LIN {X 0,Y 580.292,Z 680.195,A -85,B 0,C 180,E1 -1968.827,E2 -1968.827} C_VEL
LIN {X 0,Y 580.317,Z 680.194,A -85,B 0,C 180,E1 -1971.644,E2 -1971.644} C_VEL
LIN {X 0,Y 580.327,Z 680.195,A -85,B 0,C 180,E1 -1974.44,E2 -1974.44} C_VEL
LIN {X 0,Y 580.324,Z 680.19,A -85,B 0,C 180,E1 -1977.223,E2 -1977.223} C_VEL
LIN {X 0,Y 580.334,Z 680.194,A -85,B 0,C 180,E1 -1980,E2 -1980} C_VEL
LIN {X 0,Y 580.338,Z 680.194,A -85,B 0,C 180,E1 -1982.777,E2 -1982.777} C_VEL
LIN {X 0,Y 580.312,Z 680.192,A -85,B 0,C 180,E1 -1985.56,E2 -1985.56} C_VEL
LIN {X 0,Y 580.321,Z 680.196,A -85,B 0,C 180,E1 -1988.356,E2 -1988.356} C_VEL
LIN {X 0,Y 580.322,Z 680.194,A -85,B 0,C 180,E1 -1991.209,E2 -1991.209} C_VEL
LIN {X 0,Y 580.297,Z 680.196,A -85,B 0,C 180,E1 -1994.337,E2 -1994.337} C_VEL
LIN {X 0,Y 580.3,Z 680.203,A -85,B 0,C 180,E1 -1996.914,E2 -1996.914} C_VEL
LIN {X 0,Y 580.291,Z 680.195,A -85,B 0,C 180,E1 -1999.823,E2 -1999.823} C_VEL
LIN {X 0,Y 580.269,Z 680.204,A -85,B 0,C 180,E1 -2001.343,E2 -2001.343} C_VEL
LIN {X 0,Y 579.573,Z 680.286,A -85,B 0,C 180,E1 -2001.923,E2 -2001.923} C_VEL
LIN {X 0,Y 576.697,Z 680.647,A -85,B 0,C 180,E1 -2002.862,E2 -2002.862} C_VEL
LIN {X 0,Y 574.296,Z 680.944,A -85,B 0,C 180,E1 -2003.619,E2 -2003.619} C_VEL
LIN {X 0,Y 573.284,Z 681.066,A -85,B 0,C 180,E1 -2004.203,E2 -2004.203} C_VEL
LIN {X 0,Y 573.211,Z 681.076,A -85,B 0,C 180,E1 -2004.4,E2 -2004.4} C_VEL
LIN {X 0,Y 573.238,Z 681.079,A -85,B 0,C 180,E1 -2006.977,E2 -2006.977} C_VEL
LIN {X 0,Y 573.235,Z 681.084,A -85,B 0,C 180,E1 -2009.489,E2 -2009.489} C_VEL
LIN {X 0,Y 573.244,Z 681.072,A -85,B 0,C 180,E1 -2012.646,E2 -2012.646} C_VEL
LIN {X 0,Y 573.243,Z 681.077,A -85,B 0,C 180,E1 -2015.186,E2 -2015.186} C_VEL
LIN {X 0,Y 573.228,Z 681.083,A -85,B 0,C 180,E1 -2017.809,E2 -2017.809} C_VEL
LIN {X 0,Y 573.237,Z 681.075,A -85,B 0,C 180,E1 -2020.526,E2 -2020.526} C_VEL
LIN {X 0,Y 573.231,Z 681.077,A -85,B 0,C 180,E1 -2023.36,E2 -2023.36} C_VEL
LIN {X 0,Y 573.229,Z 681.08,A -85,B 0,C 180,E1 -2026.333,E2 -2026.333} C_VEL
LIN {X 0,Y 573.22,Z 681.08,A -85,B 0,C 180,E1 -2028.544,E2 -2028.544} C_VEL
LIN {X 0,Y 573.301,Z 681.29,A -85,B 0,C 180,E1 -2031.465,E2 -2031.465} C_VEL
LIN {X 0,Y 573.493,Z 682.25,A -85,B 0,C 180,E1 -2031.564,E2 -2031.564} C_VEL
LIN {X 0,Y 574.016,Z 685.356,A -85,B 0,C 180,E1 -2031.626,E2 -2031.626} C_VEL
LIN {X 0,Y 573.888,Z 762.761,A -85,B 0,C 180,E1 -2032.619,E2 -2032.619} C_VEL
LIN {X 0,Y 573.797,Z 776.245,A -85,B 0,C 180,E1 -2032.945,E2 -2032.945} C_VEL
LIN {X 0,Y 573.673,Z 788.533,A -85,B 0,C 180,E1 -2033.385,E2 -2033.385} C_VEL
LIN {X 0,Y 573.574,Z 800.656,A -85,B 0,C 180,E1 -2033.976,E2 -2033.976} C_VEL
LIN {X 0,Y 573.428,Z 812.525,A -85,B 0,C 180,E1 -2034.722,E2 -2034.722} C_VEL
LIN {X 0,Y 573.348,Z 822.555,A -85,B 0,C 180,E1 -2035.512,E2 -2035.512} C_VEL
LIN {X 0,Y 573.187,Z 832.534,A -85,B 0,C 180,E1 -2036.488,E2 -2036.488} C_VEL
LIN {X 0,Y 573.17,Z 839.774,A -85,B 0,C 180,E1 -2037.351,E2 -2037.351} C_VEL
LIN {X 0,Y 573.102,Z 846.922,A -85,B 0,C 180,E1 -2038.384,E2 -2038.384} C_VEL
LIN {X 0,Y 573.027,Z 853.016,A -85,B 0,C 180,E1 -2039.48,E2 -2039.48} C_VEL
LIN {X 0,Y 573.024,Z 857.961,A -85,B 0,C 180,E1 -2040.622,E2 -2040.622} C_VEL
LIN {X 0,Y 572.974,Z 860.64,A -85,B 0,C 180,E1 -2041.423,E2 -2041.423} C_VEL
LIN {X 0,Y 572.963,Z 862.779,A -85,B 0,C 180,E1 -2042.219,E2 -2042.219} C_VEL
LIN {X 0,Y 572.961,Z 865.101,A -85,B 0,C 180,E1 -2043.564,E2 -2043.564} C_VEL
LIN {X 0,Y 572.939,Z 865.901,A -85,B 0,C 180,E1 -2044.576,E2 -2044.576} C_VEL
LIN {X 0,Y 572.951,Z 865.938,A -85,B 0,C 180,E1 -2045.353,E2 -2045.353} C_VEL
LIN {X 0,Y 572.926,Z 865.53,A -85,B 0,C 180,E1 -2046.122,E2 -2046.122} C_VEL
LIN {X 0,Y 572.952,Z 864.563,A -85,B 0,C 180,E1 -2046.923,E2 -2046.923} C_VEL
LIN {X 0,Y 572.945,Z 863.24,A -85,B 0,C 180,E1 -2047.652,E2 -2047.652} C_VEL
LIN {X 0,Y 572.989,Z 860.305,A -85,B 0,C 180,E1 -2048.778,E2 -2048.778} C_VEL
LIN {X 0,Y 573.03,Z 856.166,A -85,B 0,C 180,E1 -2049.917,E2 -2049.917} C_VEL
LIN {X 0,Y 573.072,Z 850.484,A -85,B 0,C 180,E1 -2051.099,E2 -2051.099} C_VEL
LIN {X 0,Y 573.119,Z 844.051,A -85,B 0,C 180,E1 -2052.149,E2 -2052.149} C_VEL
LIN {X 0,Y 573.174,Z 836.754,A -85,B 0,C 180,E1 -2053.118,E2 -2053.118} C_VEL
LIN {X 0,Y 573.266,Z 826.991,A -85,B 0,C 180,E1 -2054.172,E2 -2054.172} C_VEL
LIN {X 0,Y 573.368,Z 817.537,A -85,B 0,C 180,E1 -2054.994,E2 -2054.994} C_VEL
LIN {X 0,Y 573.504,Z 807.239,A -85,B 0,C 180,E1 -2055.723,E2 -2055.723} C_VEL
LIN {X 0,Y 573.606,Z 796.002,A -85,B 0,C 180,E1 -2056.359,E2 -2056.359} C_VEL
LIN {X 0,Y 573.724,Z 783.527,A -85,B 0,C 180,E1 -2056.903,E2 -2056.903} C_VEL
LIN {X 0,Y 573.833,Z 770.218,A -85,B 0,C 180,E1 -2057.31,E2 -2057.31} C_VEL
LIN {X 0,Y 573.914,Z 757.259,A -85,B 0,C 180,E1 -2057.559,E2 -2057.559} C_VEL
LIN {X 0,Y 573.909,Z 683.635,A -85,B 0,C 180,E1 -2058.488,E2 -2058.488} C_VEL
LIN {X 0,Y 573.375,Z 681.682,A -85,B 0,C 180,E1 -2058.567,E2 -2058.567} C_VEL
LIN {X 0,Y 573.274,Z 681.113,A -85,B 0,C 180,E1 -2058.689,E2 -2058.689} C_VEL
LIN {X 0,Y 573.245,Z 681.078,A -85,B 0,C 180,E1 -2061.541,E2 -2061.541} C_VEL
LIN {X 0,Y 573.267,Z 681.076,A -85,B 0,C 180,E1 -2064.373,E2 -2064.373} C_VEL
LIN {X 0,Y 573.309,Z 681.071,A -85,B 0,C 180,E1 -2067.893,E2 -2067.893} C_VEL
LIN {X 0,Y 573.319,Z 681.071,A -85,B 0,C 180,E1 -2070.001,E2 -2070.001} C_VEL
LIN {X 0,Y 573.279,Z 681.072,A -85,B 0,C 180,E1 -2072.812,E2 -2072.812} C_VEL
LIN {X 0,Y 573.257,Z 681.072,A -85,B 0,C 180,E1 -2075.63,E2 -2075.63} C_VEL
LIN {X 0,Y 573.237,Z 681.084,A -85,B 0,C 180,E1 -2078.461,E2 -2078.461} C_VEL
LIN {X 0,Y 573.239,Z 681.074,A -85,B 0,C 180,E1 -2081.314,E2 -2081.314} C_VEL
LIN {X 0,Y 573.264,Z 681.076,A -85,B 0,C 180,E1 -2084.415,E2 -2084.415} C_VEL
LIN {X 0,Y 573.223,Z 681.08,A -85,B 0,C 180,E1 -2087.114,E2 -2087.114} C_VEL
LIN {X 0,Y 573.205,Z 681.076,A -85,B 0,C 180,E1 -2090.079,E2 -2090.079} C_VEL
LIN {X 0,Y 573.218,Z 681.078,A -85,B 0,C 180,E1 -2092.34,E2 -2092.34} C_VEL
LIN {X 0,Y 573.196,Z 681.081,A -85,B 0,C 180,E1 -2095.414,E2 -2095.414} C_VEL
LIN {X 0,Y 573.2,Z 681.077,A -85,B 0,C 180,E1 -2098.018,E2 -2098.018} C_VEL
LIN {X 0,Y 573.201,Z 681.083,A -85,B 0,C 180,E1 -2100.877,E2 -2100.877} C_VEL
LIN {X 0,Y 573.195,Z 681.082,A -85,B 0,C 180,E1 -2103.513,E2 -2103.513} C_VEL
LIN {X 0,Y 573.181,Z 681.079,A -85,B 0,C 180,E1 -2106.055,E2 -2106.055} C_VEL
LIN {X 0,Y 573.177,Z 681.081,A -85,B 0,C 180,E1 -2108.708,E2 -2108.708} C_VEL
LIN {X 0,Y 573.194,Z 681.089,A -85,B 0,C 180,E1 -2111.588,E2 -2111.588} C_VEL
LIN {X 0,Y 573.207,Z 681.078,A -85,B 0,C 180,E1 -2114.337,E2 -2114.337} C_VEL
LIN {X 0,Y 573.213,Z 681.081,A -85,B 0,C 180,E1 -2117.363,E2 -2117.363} C_VEL
LIN {X 0,Y 573.224,Z 681.076,A -85,B 0,C 180,E1 -2120.572,E2 -2120.572} C_VEL
LIN {X 0,Y 573.183,Z 681.081,A -85,B 0,C 180,E1 -2123.072,E2 -2123.072} C_VEL
LIN {X 0,Y 573.242,Z 681.079,A -85,B 0,C 180,E1 -2125.669,E2 -2125.669} C_VEL
LIN {X 0,Y 573.21,Z 681.087,A -85,B 0,C 180,E1 -2128.182,E2 -2128.182} C_VEL
LIN {X 0,Y 573.221,Z 681.08,A -85,B 0,C 180,E1 -2130.631,E2 -2130.631} C_VEL
LIN {X 0,Y 573.257,Z 681.217,A -85,B 0,C 180,E1 -2133.443,E2 -2133.443} C_VEL
LIN {X 0,Y 573.405,Z 682.037,A -85,B 0,C 180,E1 -2133.552,E2 -2133.552} C_VEL
LIN {X 0,Y 574.019,Z 683.936,A -85,B 0,C 180,E1 -2133.608,E2 -2133.608} C_VEL
LIN {X 0,Y 573.874,Z 761.452,A -85,B 0,C 180,E1 -2134.595,E2 -2134.595} C_VEL
LIN {X 0,Y 573.817,Z 774.103,A -85,B 0,C 180,E1 -2134.885,E2 -2134.885} C_VEL
LIN {X 0,Y 573.684,Z 785.769,A -85,B 0,C 180,E1 -2135.278,E2 -2135.278} C_VEL
LIN {X 0,Y 573.596,Z 796.622,A -85,B 0,C 180,E1 -2135.766,E2 -2135.766} C_VEL
LIN {X 0,Y 573.486,Z 806.696,A -85,B 0,C 180,E1 -2136.337,E2 -2136.337} C_VEL
LIN {X 0,Y 573.375,Z 816.262,A -85,B 0,C 180,E1 -2137.002,E2 -2137.002} C_VEL
LIN {X 0,Y 573.273,Z 826.276,A -85,B 0,C 180,E1 -2137.853,E2 -2137.853} C_VEL
LIN {X 0,Y 573.166,Z 836.526,A -85,B 0,C 180,E1 -2138.943,E2 -2138.943} C_VEL
LIN {X 0,Y 573.09,Z 843.894,A -85,B 0,C 180,E1 -2139.917,E2 -2139.917} C_VEL
LIN {X 0,Y 573.05,Z 851.003,A -85,B 0,C 180,E1 -2141.096,E2 -2141.096} C_VEL
LIN {X 0,Y 572.995,Z 856.009,A -85,B 0,C 180,E1 -2142.143,E2 -2142.143} C_VEL
LIN {X 0,Y 572.999,Z 859.538,A -85,B 0,C 180,E1 -2143.078,E2 -2143.078} C_VEL
LIN {X 0,Y 572.934,Z 863.018,A -85,B 0,C 180,E1 -2144.343,E2 -2144.343} C_VEL
LIN {X 0,Y 572.948,Z 865.26,A -85,B 0,C 180,E1 -2145.709,E2 -2145.709} C_VEL
LIN {X 0,Y 572.971,Z 865.85,A -85,B 0,C 180,E1 -2146.523,E2 -2146.523} C_VEL
LIN {X 0,Y 572.946,Z 865.962,A -85,B 0,C 180,E1 -2147.244,E2 -2147.244} C_VEL
LIN {X 0,Y 572.948,Z 865.641,A -85,B 0,C 180,E1 -2147.964,E2 -2147.964} C_VEL
LIN {X 0,Y 572.986,Z 863.757,A -85,B 0,C 180,E1 -2149.398,E2 -2149.398} C_VEL
LIN {X 0,Y 572.985,Z 861.23,A -85,B 0,C 180,E1 -2150.469,E2 -2150.469} C_VEL
LIN {X 0,Y 573.022,Z 857.69,A -85,B 0,C 180,E1 -2151.536,E2 -2151.536} C_VEL
LIN {X 0,Y 573.028,Z 853.051,A -85,B 0,C 180,E1 -2152.601,E2 -2152.601} C_VEL
LIN {X 0,Y 573.057,Z 847.179,A -85,B 0,C 180,E1 -2153.663,E2 -2153.663} C_VEL
LIN {X 0,Y 573.1,Z 839.878,A -85,B 0,C 180,E1 -2154.723,E2 -2154.723} C_VEL
LIN {X 0,Y 573.22,Z 832.446,A -85,B 0,C 180,E1 -2155.605,E2 -2155.605} C_VEL
LIN {X 0,Y 573.281,Z 825.479,A -85,B 0,C 180,E1 -2156.31,E2 -2156.31} C_VEL
LIN {X 0,Y 573.401,Z 816.075,A -85,B 0,C 180,E1 -2157.102,E2 -2157.102} C_VEL
LIN {X 0,Y 573.518,Z 805.856,A -85,B 0,C 180,E1 -2157.805,E2 -2157.805} C_VEL
LIN {X 0,Y 573.578,Z 794.739,A -85,B 0,C 180,E1 -2158.42,E2 -2158.42} C_VEL
LIN {X 0,Y 573.758,Z 783.44,A -85,B 0,C 180,E1 -2158.903,E2 -2158.903} C_VEL
LIN {X 0,Y 573.836,Z 768.97,A -85,B 0,C 180,E1 -2159.342,E2 -2159.342} C_VEL
LIN {X 0,Y 573.918,Z 755.563,A -85,B 0,C 180,E1 -2159.583,E2 -2159.583} C_VEL
LIN {X 0,Y 574.036,Z 683.885,A -85,B 0,C 180,E1 -2160.482,E2 -2160.482} C_VEL
LIN {X 0,Y 573.443,Z 681.868,A -85,B 0,C 180,E1 -2160.548,E2 -2160.548} C_VEL
LIN {X 0,Y 573.329,Z 681.115,A -85,B 0,C 180,E1 -2160.702,E2 -2160.702} C_VEL
LIN {X 0,Y 573.303,Z 681.068,A -85,B 0,C 180,E1 -2162.811,E2 -2162.811} C_VEL
LIN {X 0,Y 573.291,Z 681.072,A -85,B 0,C 180,E1 -2165.628,E2 -2165.628} C_VEL
LIN {X 0,Y 573.259,Z 681.077,A -85,B 0,C 180,E1 -2168.46,E2 -2168.46} C_VEL
LIN {X 0,Y 573.279,Z 681.069,A -85,B 0,C 180,E1 -2171.312,E2 -2171.312} C_VEL
LIN {X 0,Y 573.288,Z 681.077,A -85,B 0,C 180,E1 -2174.424,E2 -2174.424} C_VEL
LIN {X 0,Y 573.262,Z 681.072,A -85,B 0,C 180,E1 -2177.111,E2 -2177.111} C_VEL
LIN {X 0,Y 573.247,Z 681.076,A -85,B 0,C 180,E1 -2180.077,E2 -2180.077} C_VEL
LIN {X 0,Y 573.237,Z 681.08,A -85,B 0,C 180,E1 -2182.338,E2 -2182.338} C_VEL
LIN {X 0,Y 573.252,Z 681.073,A -85,B 0,C 180,E1 -2185.41,E2 -2185.41} C_VEL
LIN {X 0,Y 573.234,Z 681.081,A -85,B 0,C 180,E1 -2188.565,E2 -2188.565} C_VEL
LIN {X 0,Y 573.23,Z 681.083,A -85,B 0,C 180,E1 -2190.993,E2 -2190.993} C_VEL
LIN {X 0,Y 573.247,Z 681.075,A -85,B 0,C 180,E1 -2193.52,E2 -2193.52} C_VEL
LIN {X 0,Y 573.22,Z 681.076,A -85,B 0,C 180,E1 -2196.051,E2 -2196.051} C_VEL
LIN {X 0,Y 573.244,Z 681.077,A -85,B 0,C 180,E1 -2198.702,E2 -2198.702} C_VEL
LIN {X 0,Y 573.233,Z 681.079,A -85,B 0,C 180,E1 -2201.592,E2 -2201.592} C_VEL
LIN {X 0,Y 573.228,Z 681.075,A -85,B 0,C 180,E1 -2204.334,E2 -2204.334} C_VEL
LIN {X 0,Y 573.245,Z 681.083,A -85,B 0,C 180,E1 -2207.358,E2 -2207.358} C_VEL
LIN {X 0,Y 573.241,Z 681.073,A -85,B 0,C 180,E1 -2210.391,E2 -2210.391} C_VEL
LIN {X 0,Y 573.238,Z 681.076,A -85,B 0,C 180,E1 -2213.075,E2 -2213.075} C_VEL
LIN {X 0,Y 573.26,Z 681.081,A -85,B 0,C 180,E1 -2215.67,E2 -2215.67} C_VEL
LIN {X 0,Y 573.245,Z 681.078,A -85,B 0,C 180,E1 -2218.184,E2 -2218.184} C_VEL
LIN {X 0,Y 573.265,Z 681.074,A -85,B 0,C 180,E1 -2220.633,E2 -2220.633} C_VEL
LIN {X 0,Y 573.257,Z 681.272,A -85,B 0,C 180,E1 -2222.629,E2 -2222.629} C_VEL
LIN {X 0,Y 574.935,Z 688.635,A -85,B 0,C 180,E1 -2223.592,E2 -2223.592} C_VEL
LIN {X 0,Y 574.576,Z 711.379,A -85,B 0,C 180,E1 -2226.193,E2 -2226.193} C_VEL
LIN {X 0,Y 574.209,Z 738.275,A -85,B 0,C 180,E1 -2229.209,E2 -2229.209} C_VEL
LIN {X 0,Y 573.871,Z 765.171,A -85,B 0,C 180,E1 -2232.171,E2 -2232.171} C_VEL
LIN {X 0,Y 573.599,Z 792.067,A -85,B 0,C 180,E1 -2235.089,E2 -2235.089} C_VEL
LIN {X 0,Y 573.536,Z 801.874,A -85,B 0,C 180,E1 -2236.129,E2 -2236.129} C_VEL
LIN {X 0,Y 574.037,Z 807.642,A -85,B 0,C 180,E1 -2236.232,E2 -2236.232} C_VEL
LIN {X 0,Y 573.876,Z 911.896,A -85,B 0,C 180,E1 -2237.556,E2 -2237.556} C_VEL
LIN {X 0,Y 573.832,Z 924.424,A -85,B 0,C 180,E1 -2237.847,E2 -2237.847} C_VEL
LIN {X 0,Y 573.708,Z 936.891,A -85,B 0,C 180,E1 -2238.275,E2 -2238.275} C_VEL
LIN {X 0,Y 573.612,Z 948.42,A -85,B 0,C 180,E1 -2238.809,E2 -2238.809} C_VEL
LIN {X 0,Y 573.475,Z 959.899,A -85,B 0,C 180,E1 -2239.496,E2 -2239.496} C_VEL
LIN {X 0,Y 573.345,Z 970.527,A -85,B 0,C 180,E1 -2240.296,E2 -2240.296} C_VEL
LIN {X 0,Y 573.238,Z 980.036,A -85,B 0,C 180,E1 -2241.184,E2 -2241.184} C_VEL
LIN {X 0,Y 573.161,Z 987.952,A -85,B 0,C 180,E1 -2242.07,E2 -2242.07} C_VEL
LIN {X 0,Y 573.076,Z 995.935,A -85,B 0,C 180,E1 -2243.183,E2 -2243.183} C_VEL
LIN {X 0,Y 573.07,Z 1002.675,A -85,B 0,C 180,E1 -2244.369,E2 -2244.369} C_VEL
LIN {X 0,Y 573.028,Z 1007.368,A -85,B 0,C 180,E1 -2245.426,E2 -2245.426} C_VEL
LIN {X 0,Y 573.022,Z 1010.954,A -85,B 0,C 180,E1 -2246.483,E2 -2246.483} C_VEL
LIN {X 0,Y 572.959,Z 1012.806,A -85,B 0,C 180,E1 -2247.187,E2 -2247.187} C_VEL
LIN {X 0,Y 572.938,Z 1014.198,A -85,B 0,C 180,E1 -2247.89,E2 -2247.89} C_VEL
LIN {X 0,Y 572.94,Z 1015.784,A -85,B 0,C 180,E1 -2249.296,E2 -2249.296} C_VEL
LIN {X 0,Y 572.938,Z 1016,A -85,B 0,C 180,E1 -2249.999,E2 -2249.999} C_VEL
LIN {X 0,Y 572.946,Z 1015.187,A -85,B 0,C 180,E1 -2251.405,E2 -2251.405} C_VEL
LIN {X 0,Y 572.938,Z 1014.202,A -85,B 0,C 180,E1 -2252.108,E2 -2252.108} C_VEL
LIN {X 0,Y 572.959,Z 1012.812,A -85,B 0,C 180,E1 -2252.811,E2 -2252.811} C_VEL
LIN {X 0,Y 573.014,Z 1009.899,A -85,B 0,C 180,E1 -2253.867,E2 -2253.867} C_VEL
LIN {X 0,Y 572.962,Z 1005.954,A -85,B 0,C 180,E1 -2254.925,E2 -2254.925} C_VEL
LIN {X 0,Y 573.067,Z 999.883,A -85,B 0,C 180,E1 -2256.159,E2 -2256.159} C_VEL
LIN {X 0,Y 573.118,Z 993.245,A -85,B 0,C 180,E1 -2257.22,E2 -2257.22} C_VEL
LIN {X 0,Y 573.191,Z 985,A -85,B 0,C 180,E1 -2258.282,E2 -2258.282} C_VEL
LIN {X 0,Y 573.319,Z 974.613,A -85,B 0,C 180,E1 -2259.347,E2 -2259.347} C_VEL
LIN {X 0,Y 573.43,Z 964.943,A -85,B 0,C 180,E1 -2260.146,E2 -2260.146} C_VEL
LIN {X 0,Y 573.552,Z 954.369,A -85,B 0,C 180,E1 -2260.857,E2 -2260.857} C_VEL
LIN {X 0,Y 573.685,Z 942.023,A -85,B 0,C 180,E1 -2261.504,E2 -2261.504} C_VEL
LIN {X 0,Y 573.737,Z 930.208,A -85,B 0,C 180,E1 -2261.973,E2 -2261.973} C_VEL
LIN {X 0,Y 573.842,Z 917.568,A -85,B 0,C 180,E1 -2262.33,E2 -2262.33} C_VEL
LIN {X 0,Y 573.946,Z 904.402,A -85,B 0,C 180,E1 -2262.552,E2 -2262.552} C_VEL
LIN {X 0,Y 573.986,Z 805.242,A -85,B 0,C 180,E1 -2263.8,E2 -2263.8} C_VEL
LIN {X 0,Y 573.534,Z 801.904,A -85,B 0,C 180,E1 -2263.869,E2 -2263.869} C_VEL
LIN {X 0,Y 573.769,Z 775.277,A -85,B 0,C 180,E1 -2266.728,E2 -2266.728} C_VEL
LIN {X 0,Y 574.121,Z 746.574,A -85,B 0,C 180,E1 -2269.871,E2 -2269.871} C_VEL
LIN {X 0,Y 574.399,Z 721.485,A -85,B 0,C 180,E1 -2272.668,E2 -2272.668} C_VEL
LIN {X 0,Y 574.808,Z 699.068,A -85,B 0,C 180,E1 -2275.207,E2 -2275.207} C_VEL
LIN {X 0,Y 574.941,Z 688.649,A -85,B 0,C 180,E1 -2276.406,E2 -2276.406} C_VEL
LIN {X 0,Y 573.258,Z 681.194,A -85,B 0,C 180,E1 -2277.394,E2 -2277.394} C_VEL
LIN {X 0,Y 573.243,Z 681.082,A -85,B 0,C 180,E1 -2280.175,E2 -2280.175} C_VEL
LIN {X 0,Y 573.249,Z 681.078,A -85,B 0,C 180,E1 -2282.644,E2 -2282.644} C_VEL
LIN {X 0,Y 573.201,Z 681.079,A -85,B 0,C 180,E1 -2285.187,E2 -2285.187} C_VEL
LIN {X 0,Y 573.228,Z 681.076,A -85,B 0,C 180,E1 -2287.806,E2 -2287.806} C_VEL
LIN {X 0,Y 573.237,Z 681.083,A -85,B 0,C 180,E1 -2290.524,E2 -2290.524} C_VEL
LIN {X 0,Y 573.232,Z 681.075,A -85,B 0,C 180,E1 -2293.358,E2 -2293.358} C_VEL
LIN {X 0,Y 573.248,Z 681.075,A -85,B 0,C 180,E1 -2296.329,E2 -2296.329} C_VEL
LIN {X 0,Y 573.266,Z 681.071,A -85,B 0,C 180,E1 -2299.477,E2 -2299.477} C_VEL
LIN {X 0,Y 573.228,Z 681.075,A -85,B 0,C 180,E1 -2302.192,E2 -2302.192} C_VEL
LIN {X 0,Y 573.259,Z 681.075,A -85,B 0,C 180,E1 -2304.816,E2 -2304.816} C_VEL
LIN {X 0,Y 573.244,Z 681.081,A -85,B 0,C 180,E1 -2307.354,E2 -2307.354} C_VEL
LIN {X 0,Y 573.243,Z 681.073,A -85,B 0,C 180,E1 -2310.51,E2 -2310.51} C_VEL
LIN {X 0,Y 573.253,Z 681.076,A -85,B 0,C 180,E1 -2313.024,E2 -2313.024} C_VEL
LIN {X 0,Y 573.264,Z 681.079,A -85,B 0,C 180,E1 -2315.366,E2 -2315.366} C_VEL
LIN {X 0,Y 573.218,Z 681.075,A -85,B 0,C 180,E1 -2318.419,E2 -2318.419} C_VEL
LIN {X 0,Y 573.266,Z 681.07,A -85,B 0,C 180,E1 -2320.728,E2 -2320.728} C_VEL
LIN {X 0,Y 573.235,Z 681.081,A -85,B 0,C 180,E1 -2323.621,E2 -2323.621} C_VEL
LIN {X 0,Y 573.262,Z 681.081,A -85,B 0,C 180,E1 -2325.807,E2 -2325.807} C_VEL
LIN {X 0,Y 573.25,Z 681.072,A -85,B 0,C 180,E1 -2328.745,E2 -2328.745} C_VEL
LIN {X 0,Y 573.273,Z 681.07,A -85,B 0,C 180,E1 -2331.54,E2 -2331.54} C_VEL
LIN {X 0,Y 573.293,Z 681.073,A -85,B 0,C 180,E1 -2334.372,E2 -2334.372} C_VEL
LIN {X 0,Y 573.292,Z 681.066,A -85,B 0,C 180,E1 -2337.189,E2 -2337.189} C_VEL
LIN {X 0,Y 573.304,Z 681.069,A -85,B 0,C 180,E1 -2340,E2 -2340} C_VEL
LIN {X 0,Y 573.303,Z 681.07,A -85,B 0,C 180,E1 -2342.811,E2 -2342.811} C_VEL
LIN {X 0,Y 573.278,Z 681.068,A -85,B 0,C 180,E1 -2345.628,E2 -2345.628} C_VEL
LIN {X 0,Y 573.278,Z 681.076,A -85,B 0,C 180,E1 -2348.46,E2 -2348.46} C_VEL
LIN {X 0,Y 573.288,Z 681.069,A -85,B 0,C 180,E1 -2351.312,E2 -2351.312} C_VEL
LIN {X 0,Y 573.264,Z 681.074,A -85,B 0,C 180,E1 -2354.423,E2 -2354.423} C_VEL
LIN {X 0,Y 573.246,Z 681.081,A -85,B 0,C 180,E1 -2357.112,E2 -2357.112} C_VEL
LIN {X 0,Y 573.238,Z 681.073,A -85,B 0,C 180,E1 -2360.077,E2 -2360.077} C_VEL
LIN {X 0,Y 573.224,Z 681.084,A -85,B 0,C 180,E1 -2363.1,E2 -2363.1} C_VEL
LIN {X 0,Y 573.211,Z 681.076,A -85,B 0,C 180,E1 -2364.4,E2 -2364.4} C_VEL
LIN {X 0,Y 572.573,Z 681.162,A -85,B 0,C 180,E1 -2364.987,E2 -2364.987} C_VEL
LIN {X 0,Y 569.74,Z 681.521,A -85,B 0,C 180,E1 -2365.938,E2 -2365.938} C_VEL
LIN {X 0,Y 567.325,Z 681.825,A -85,B 0,C 180,E1 -2366.704,E2 -2366.704} C_VEL
LIN {X 0,Y 566.279,Z 681.951,A -85,B 0,C 180,E1 -2367.296,E2 -2367.296} C_VEL
LIN {X 0,Y 566.191,Z 681.958,A -85,B 0,C 180,E1 -2367.496,E2 -2367.496} C_VEL
LIN {X 0,Y 566.19,Z 681.957,A -85,B 0,C 180,E1 -2369.77,E2 -2369.77} C_VEL
LIN {X 0,Y 566.194,Z 681.95,A -85,B 0,C 180,E1 -2372.431,E2 -2372.431} C_VEL
LIN {X 0,Y 566.191,Z 681.953,A -85,B 0,C 180,E1 -2374.993,E2 -2374.993} C_VEL
LIN {X 0,Y 566.188,Z 681.959,A -85,B 0,C 180,E1 -2377.462,E2 -2377.462} C_VEL
LIN {X 0,Y 566.199,Z 681.955,A -85,B 0,C 180,E1 -2380.2,E2 -2380.2} C_VEL
LIN {X 0,Y 566.194,Z 681.951,A -85,B 0,C 180,E1 -2383.055,E2 -2383.055} C_VEL
LIN {X 0,Y 566.187,Z 681.96,A -85,B 0,C 180,E1 -2386.051,E2 -2386.051} C_VEL
LIN {X 0,Y 566.198,Z 681.953,A -85,B 0,C 180,E1 -2389.216,E2 -2389.216} C_VEL
LIN {X 0,Y 566.254,Z 682.179,A -85,B 0,C 180,E1 -2391.306,E2 -2391.306} C_VEL
LIN {X 0,Y 566.569,Z 683.524,A -85,B 0,C 180,E1 -2391.42,E2 -2391.42} C_VEL
LIN {X 0,Y 567.115,Z 685.653,A -85,B 0,C 180,E1 -2391.463,E2 -2391.463} C_VEL
LIN {X 0,Y 566.971,Z 762.537,A -85,B 0,C 180,E1 -2392.46,E2 -2392.46} C_VEL
LIN {X 0,Y 566.859,Z 776.007,A -85,B 0,C 180,E1 -2392.787,E2 -2392.787} C_VEL
LIN {X 0,Y 566.736,Z 787.432,A -85,B 0,C 180,E1 -2393.195,E2 -2393.195} C_VEL
LIN {X 0,Y 566.625,Z 798.688,A -85,B 0,C 180,E1 -2393.728,E2 -2393.728} C_VEL
LIN {X 0,Y 566.498,Z 810.11,A -85,B 0,C 180,E1 -2394.425,E2 -2394.425} C_VEL
LIN {X 0,Y 566.311,Z 820.193,A -85,B 0,C 180,E1 -2395.191,E2 -2395.191} C_VEL
LIN {X 0,Y 566.213,Z 829.39,A -85,B 0,C 180,E1 -2396.046,E2 -2396.046} C_VEL
LIN {X 0,Y 566.05,Z 838.458,A -85,B 0,C 180,E1 -2397.08,E2 -2397.08} C_VEL
LIN {X 0,Y 566.041,Z 845.999,A -85,B 0,C 180,E1 -2398.152,E2 -2398.152} C_VEL
LIN {X 0,Y 565.956,Z 852.941,A -85,B 0,C 180,E1 -2399.395,E2 -2399.395} C_VEL
LIN {X 0,Y 565.93,Z 858.454,A -85,B 0,C 180,E1 -2400.708,E2 -2400.708} C_VEL
LIN {X 0,Y 565.868,Z 861.979,A -85,B 0,C 180,E1 -2401.862,E2 -2401.862} C_VEL
LIN {X 0,Y 565.844,Z 863.724,A -85,B 0,C 180,E1 -2402.643,E2 -2402.643} C_VEL
LIN {X 0,Y 565.856,Z 864.984,A -85,B 0,C 180,E1 -2403.442,E2 -2403.442} C_VEL
LIN {X 0,Y 565.829,Z 865.72,A -85,B 0,C 180,E1 -2404.234,E2 -2404.234} C_VEL
LIN {X 0,Y 565.838,Z 866,A -85,B 0,C 180,E1 -2405.054,E2 -2405.054} C_VEL
LIN {X 0,Y 565.825,Z 865.754,A -85,B 0,C 180,E1 -2405.804,E2 -2405.804} C_VEL
LIN {X 0,Y 565.833,Z 864.79,A -85,B 0,C 180,E1 -2406.8,E2 -2406.8} C_VEL
LIN {X 0,Y 565.854,Z 862.235,A -85,B 0,C 180,E1 -2408.125,E2 -2408.125} C_VEL
LIN {X 0,Y 565.898,Z 858.838,A -85,B 0,C 180,E1 -2409.272,E2 -2409.272} C_VEL
LIN {X 0,Y 565.973,Z 854.261,A -85,B 0,C 180,E1 -2410.412,E2 -2410.412} C_VEL
LIN {X 0,Y 565.988,Z 848.418,A -85,B 0,C 180,E1 -2411.541,E2 -2411.541} C_VEL
LIN {X 0,Y 566.061,Z 841.064,A -85,B 0,C 180,E1 -2412.665,E2 -2412.665} C_VEL
LIN {X 0,Y 566.194,Z 831.852,A -85,B 0,C 180,E1 -2413.784,E2 -2413.784} C_VEL
LIN {X 0,Y 566.267,Z 822.433,A -85,B 0,C 180,E1 -2414.709,E2 -2414.709} C_VEL
LIN {X 0,Y 566.408,Z 811.869,A -85,B 0,C 180,E1 -2415.544,E2 -2415.544} C_VEL
LIN {X 0,Y 566.593,Z 800.19,A -85,B 0,C 180,E1 -2416.278,E2 -2416.278} C_VEL
LIN {X 0,Y 566.733,Z 787.92,A -85,B 0,C 180,E1 -2416.875,E2 -2416.875} C_VEL
LIN {X 0,Y 566.879,Z 774.93,A -85,B 0,C 180,E1 -2417.334,E2 -2417.334} C_VEL
LIN {X 0,Y 566.952,Z 762.486,A -85,B 0,C 180,E1 -2417.631,E2 -2417.631} C_VEL
LIN {X 0,Y 567.037,Z 685.043,A -85,B 0,C 180,E1 -2418.636,E2 -2418.636} C_VEL
LIN {X 0,Y 566.368,Z 682.687,A -85,B 0,C 180,E1 -2418.714,E2 -2418.714} C_VEL
LIN {X 0,Y 566.215,Z 682.009,A -85,B 0,C 180,E1 -2418.84,E2 -2418.84} C_VEL
LIN {X 0,Y 566.196,Z 681.956,A -85,B 0,C 180,E1 -2421.435,E2 -2421.435} C_VEL
LIN {X 0,Y 566.238,Z 681.953,A -85,B 0,C 180,E1 -2424.303,E2 -2424.303} C_VEL
LIN {X 0,Y 566.279,Z 681.947,A -85,B 0,C 180,E1 -2427.867,E2 -2427.867} C_VEL
LIN {X 0,Y 566.288,Z 681.947,A -85,B 0,C 180,E1 -2430.001,E2 -2430.001} C_VEL
LIN {X 0,Y 566.245,Z 681.948,A -85,B 0,C 180,E1 -2432.847,E2 -2432.847} C_VEL
LIN {X 0,Y 566.228,Z 681.948,A -85,B 0,C 180,E1 -2435.7,E2 -2435.7} C_VEL
LIN {X 0,Y 566.19,Z 681.962,A -85,B 0,C 180,E1 -2438.567,E2 -2438.567} C_VEL
LIN {X 0,Y 566.195,Z 681.951,A -85,B 0,C 180,E1 -2441.456,E2 -2441.456} C_VEL
LIN {X 0,Y 566.219,Z 681.955,A -85,B 0,C 180,E1 -2444.498,E2 -2444.498} C_VEL
LIN {X 0,Y 566.176,Z 681.955,A -85,B 0,C 180,E1 -2447.333,E2 -2447.333} C_VEL
LIN {X 0,Y 566.178,Z 681.951,A -85,B 0,C 180,E1 -2449.583,E2 -2449.583} C_VEL
LIN {X 0,Y 566.187,Z 681.952,A -85,B 0,C 180,E1 -2451.864,E2 -2451.864} C_VEL
LIN {X 0,Y 566.152,Z 681.956,A -85,B 0,C 180,E1 -2454.184,E2 -2454.184} C_VEL
LIN {X 0,Y 566.165,Z 681.956,A -85,B 0,C 180,E1 -2456.649,E2 -2456.649} C_VEL
LIN {X 0,Y 566.141,Z 681.96,A -85,B 0,C 180,E1 -2459.66,E2 -2459.66} C_VEL
LIN {X 0,Y 566.176,Z 681.953,A -85,B 0,C 180,E1 -2462.425,E2 -2462.425} C_VEL
LIN {X 0,Y 566.152,Z 681.957,A -85,B 0,C 180,E1 -2464.985,E2 -2464.985} C_VEL
LIN {X 0,Y 566.182,Z 681.962,A -85,B 0,C 180,E1 -2467.463,E2 -2467.463} C_VEL
LIN {X 0,Y 566.161,Z 681.956,A -85,B 0,C 180,E1 -2470.204,E2 -2470.204} C_VEL
LIN {X 0,Y 566.137,Z 681.961,A -85,B 0,C 180,E1 -2473.061,E2 -2473.061} C_VEL
LIN {X 0,Y 566.14,Z 681.962,A -85,B 0,C 180,E1 -2476.056,E2 -2476.056} C_VEL
LIN {X 0,Y 566.134,Z 681.959,A -85,B 0,C 180,E1 -2478.856,E2 -2478.856} C_VEL
LIN {X 0,Y 566.158,Z 681.96,A -85,B 0,C 180,E1 -2481.45,E2 -2481.45} C_VEL
LIN {X 0,Y 566.135,Z 681.963,A -85,B 0,C 180,E1 -2484.306,E2 -2484.306} C_VEL
LIN {X 0,Y 566.165,Z 681.956,A -85,B 0,C 180,E1 -2486.894,E2 -2486.894} C_VEL
LIN {X 0,Y 566.161,Z 681.958,A -85,B 0,C 180,E1 -2489.406,E2 -2489.406} C_VEL
LIN {X 0,Y 566.133,Z 681.966,A -85,B 0,C 180,E1 -2491.853,E2 -2491.853} C_VEL
LIN {X 0,Y 566.195,Z 682.159,A -85,B 0,C 180,E1 -2493.297,E2 -2493.297} C_VEL
LIN {X 0,Y 566.489,Z 683.306,A -85,B 0,C 180,E1 -2493.414,E2 -2493.414} C_VEL
LIN {X 0,Y 567.125,Z 685.465,A -85,B 0,C 180,E1 -2493.461,E2 -2493.461} C_VEL
LIN {X 0,Y 566.962,Z 761.993,A -85,B 0,C 180,E1 -2494.452,E2 -2494.452} C_VEL
LIN {X 0,Y 566.853,Z 773.749,A -85,B 0,C 180,E1 -2494.723,E2 -2494.723} C_VEL
LIN {X 0,Y 566.74,Z 785.24,A -85,B 0,C 180,E1 -2495.111,E2 -2495.111} C_VEL
LIN {X 0,Y 566.611,Z 795.056,A -85,B 0,C 180,E1 -2495.545,E2 -2495.545} C_VEL
LIN {X 0,Y 566.532,Z 805.456,A -85,B 0,C 180,E1 -2496.126,E2 -2496.126} C_VEL
LIN {X 0,Y 566.385,Z 815.224,A -85,B 0,C 180,E1 -2496.798,E2 -2496.798} C_VEL
LIN {X 0,Y 566.291,Z 824.388,A -85,B 0,C 180,E1 -2497.565,E2 -2497.565} C_VEL
LIN {X 0,Y 566.166,Z 832.923,A -85,B 0,C 180,E1 -2498.43,E2 -2498.43} C_VEL
LIN {X 0,Y 566.069,Z 839.916,A -85,B 0,C 180,E1 -2499.277,E2 -2499.277} C_VEL
LIN {X 0,Y 566.033,Z 847.603,A -85,B 0,C 180,E1 -2500.413,E2 -2500.413} C_VEL
LIN {X 0,Y 565.944,Z 853.639,A -85,B 0,C 180,E1 -2501.538,E2 -2501.538} C_VEL
LIN {X 0,Y 565.901,Z 858.292,A -85,B 0,C 180,E1 -2502.659,E2 -2502.659} C_VEL
LIN {X 0,Y 565.883,Z 860.707,A -85,B 0,C 180,E1 -2503.402,E2 -2503.402} C_VEL
LIN {X 0,Y 565.833,Z 862.637,A -85,B 0,C 180,E1 -2504.142,E2 -2504.142} C_VEL
LIN {X 0,Y 565.814,Z 864.153,A -85,B 0,C 180,E1 -2504.88,E2 -2504.88} C_VEL
LIN {X 0,Y 565.857,Z 865.208,A -85,B 0,C 180,E1 -2505.645,E2 -2505.645} C_VEL
LIN {X 0,Y 565.845,Z 865.997,A -85,B 0,C 180,E1 -2507.081,E2 -2507.081} C_VEL
LIN {X 0,Y 565.868,Z 865.74,A -85,B 0,C 180,E1 -2507.811,E2 -2507.811} C_VEL
LIN {X 0,Y 565.895,Z 864.072,A -85,B 0,C 180,E1 -2509.264,E2 -2509.264} C_VEL
LIN {X 0,Y 565.875,Z 860.645,A -85,B 0,C 180,E1 -2510.708,E2 -2510.708} C_VEL
LIN {X 0,Y 565.932,Z 856.906,A -85,B 0,C 180,E1 -2511.789,E2 -2511.789} C_VEL
LIN {X 0,Y 565.971,Z 852.049,A -85,B 0,C 180,E1 -2512.867,E2 -2512.867} C_VEL
LIN {X 0,Y 566.011,Z 845.938,A -85,B 0,C 180,E1 -2513.941,E2 -2513.941} C_VEL
LIN {X 0,Y 566.045,Z 839.743,A -85,B 0,C 180,E1 -2514.835,E2 -2514.835} C_VEL
LIN {X 0,Y 566.169,Z 832.292,A -85,B 0,C 180,E1 -2515.729,E2 -2515.729} C_VEL
LIN {X 0,Y 566.238,Z 825.301,A -85,B 0,C 180,E1 -2516.442,E2 -2516.442} C_VEL
LIN {X 0,Y 566.382,Z 815.853,A -85,B 0,C 180,E1 -2517.244,E2 -2517.244} C_VEL
LIN {X 0,Y 566.511,Z 806.994,A -85,B 0,C 180,E1 -2517.867,E2 -2517.867} C_VEL
LIN {X 0,Y 566.557,Z 797.875,A -85,B 0,C 180,E1 -2518.401,E2 -2518.401} C_VEL
LIN {X 0,Y 566.742,Z 787.43,A -85,B 0,C 180,E1 -2518.89,E2 -2518.89} C_VEL
LIN {X 0,Y 566.86,Z 776.289,A -85,B 0,C 180,E1 -2519.29,E2 -2519.29} C_VEL
LIN {X 0,Y 566.911,Z 765.004,A -85,B 0,C 180,E1 -2519.578,E2 -2519.578} C_VEL
LIN {X 0,Y 567.006,Z 750.73,A -85,B 0,C 180,E1 -2519.8,E2 -2519.8} C_VEL
LIN {X 0,Y 567.146,Z 685.161,A -85,B 0,C 180,E1 -2520.632,E2 -2520.632} C_VEL
LIN {X 0,Y 566.414,Z 682.703,A -85,B 0,C 180,E1 -2520.711,E2 -2520.711} C_VEL
LIN {X 0,Y 566.283,Z 682.003,A -85,B 0,C 180,E1 -2520.844,E2 -2520.844} C_VEL
LIN {X 0,Y 566.271,Z 681.945,A -85,B 0,C 180,E1 -2522.845,E2 -2522.845} C_VEL
LIN {X 0,Y 566.258,Z 681.95,A -85,B 0,C 180,E1 -2525.698,E2 -2525.698} C_VEL
LIN {X 0,Y 566.21,Z 681.954,A -85,B 0,C 180,E1 -2528.566,E2 -2528.566} C_VEL
LIN {X 0,Y 566.249,Z 681.945,A -85,B 0,C 180,E1 -2531.454,E2 -2531.454} C_VEL
LIN {X 0,Y 566.241,Z 681.954,A -85,B 0,C 180,E1 -2534.506,E2 -2534.506} C_VEL
LIN {X 0,Y 566.2,Z 681.951,A -85,B 0,C 180,E1 -2537.332,E2 -2537.332} C_VEL
LIN {X 0,Y 566.213,Z 681.957,A -85,B 0,C 180,E1 -2540.337,E2 -2540.337} C_VEL
LIN {X 0,Y 566.174,Z 681.955,A -85,B 0,C 180,E1 -2543.28,E2 -2543.28} C_VEL
LIN {X 0,Y 566.213,Z 681.949,A -85,B 0,C 180,E1 -2545.749,E2 -2545.749} C_VEL
LIN {X 0,Y 566.193,Z 681.96,A -85,B 0,C 180,E1 -2548.953,E2 -2548.953} C_VEL
LIN {X 0,Y 566.198,Z 681.953,A -85,B 0,C 180,E1 -2551.422,E2 -2551.422} C_VEL
LIN {X 0,Y 566.204,Z 681.95,A -85,B 0,C 180,E1 -2553.956,E2 -2553.956} C_VEL
LIN {X 0,Y 566.205,Z 681.953,A -85,B 0,C 180,E1 -2556.57,E2 -2556.57} C_VEL
LIN {X 0,Y 566.219,Z 681.951,A -85,B 0,C 180,E1 -2559.685,E2 -2559.685} C_VEL
LIN {X 0,Y 566.208,Z 681.955,A -85,B 0,C 180,E1 -2562.917,E2 -2562.917} C_VEL
LIN {X 0,Y 566.2,Z 681.952,A -85,B 0,C 180,E1 -2566.049,E2 -2566.049} C_VEL
LIN {X 0,Y 566.209,Z 681.956,A -85,B 0,C 180,E1 -2569.214,E2 -2569.214} C_VEL
LIN {X 0,Y 566.187,Z 681.961,A -85,B 0,C 180,E1 -2571.636,E2 -2571.636} C_VEL
LIN {X 0,Y 566.155,Z 681.958,A -85,B 0,C 180,E1 -2574.306,E2 -2574.306} C_VEL
LIN {X 0,Y 566.206,Z 681.951,A -85,B 0,C 180,E1 -2576.896,E2 -2576.896} C_VEL
LIN {X 0,Y 566.185,Z 681.959,A -85,B 0,C 180,E1 -2579.407,E2 -2579.407} C_VEL
LIN {X 0,Y 566.229,Z 682.124,A -85,B 0,C 180,E1 -2582.36,E2 -2582.36} C_VEL
LIN {X 0,Y 568.127,Z 689.997,A -85,B 0,C 180,E1 -2583.412,E2 -2583.412} C_VEL
LIN {X 0,Y 567.842,Z 706.336,A -85,B 0,C 180,E1 -2585.309,E2 -2585.309} C_VEL
LIN {X 0,Y 567.499,Z 728.189,A -85,B 0,C 180,E1 -2587.807,E2 -2587.807} C_VEL
LIN {X 0,Y 567.141,Z 753.404,A -85,B 0,C 180,E1 -2590.64,E2 -2590.64} C_VEL
LIN {X 0,Y 566.756,Z 780.3,A -85,B 0,C 180,E1 -2593.613,E2 -2593.613} C_VEL
LIN {X 0,Y 566.534,Z 801.872,A -85,B 0,C 180,E1 -2595.954,E2 -2595.954} C_VEL
LIN {X 0,Y 567.16,Z 807.642,A -85,B 0,C 180,E1 -2596.062,E2 -2596.062} C_VEL
LIN {X 0,Y 566.96,Z 911.896,A -85,B 0,C 180,E1 -2597.402,E2 -2597.402} C_VEL
LIN {X 0,Y 566.891,Z 925.186,A -85,B 0,C 180,E1 -2597.719,E2 -2597.719} C_VEL
LIN {X 0,Y 566.757,Z 936.892,A -85,B 0,C 180,E1 -2598.129,E2 -2598.129} C_VEL
LIN {X 0,Y 566.629,Z 949.144,A -85,B 0,C 180,E1 -2598.708,E2 -2598.708} C_VEL
LIN {X 0,Y 566.461,Z 961.189,A -85,B 0,C 180,E1 -2599.454,E2 -2599.454} C_VEL
LIN {X 0,Y 566.32,Z 971.588,A -85,B 0,C 180,E1 -2600.264,E2 -2600.264} C_VEL
LIN {X 0,Y 566.206,Z 980.046,A -85,B 0,C 180,E1 -2601.073,E2 -2601.073} C_VEL
LIN {X 0,Y 566.112,Z 987.952,A -85,B 0,C 180,E1 -2601.971,E2 -2601.971} C_VEL
LIN {X 0,Y 566.005,Z 995.615,A -85,B 0,C 180,E1 -2603.046,E2 -2603.046} C_VEL
LIN {X 0,Y 566.004,Z 1002.675,A -85,B 0,C 180,E1 -2604.298,E2 -2604.298} C_VEL
LIN {X 0,Y 565.933,Z 1007.368,A -85,B 0,C 180,E1 -2605.369,E2 -2605.369} C_VEL
LIN {X 0,Y 565.927,Z 1010.954,A -85,B 0,C 180,E1 -2606.439,E2 -2606.439} C_VEL
LIN {X 0,Y 565.878,Z 1012.806,A -85,B 0,C 180,E1 -2607.151,E2 -2607.151} C_VEL
LIN {X 0,Y 565.839,Z 1014.197,A -85,B 0,C 180,E1 -2607.864,E2 -2607.864} C_VEL
LIN {X 0,Y 565.841,Z 1015.784,A -85,B 0,C 180,E1 -2609.287,E2 -2609.287} C_VEL
LIN {X 0,Y 565.839,Z 1016,A -85,B 0,C 180,E1 -2609.999,E2 -2609.999} C_VEL
LIN {X 0,Y 565.845,Z 1015.187,A -85,B 0,C 180,E1 -2611.422,E2 -2611.422} C_VEL
LIN {X 0,Y 565.839,Z 1014.202,A -85,B 0,C 180,E1 -2612.134,E2 -2612.134} C_VEL
LIN {X 0,Y 565.877,Z 1012.812,A -85,B 0,C 180,E1 -2612.846,E2 -2612.846} C_VEL
LIN {X 0,Y 565.926,Z 1009.899,A -85,B 0,C 180,E1 -2613.915,E2 -2613.915} C_VEL
LIN {X 0,Y 565.877,Z 1005.953,A -85,B 0,C 180,E1 -2614.986,E2 -2614.986} C_VEL
LIN {X 0,Y 565.994,Z 999.883,A -85,B 0,C 180,E1 -2616.236,E2 -2616.236} C_VEL
LIN {X 0,Y 566.051,Z 993.245,A -85,B 0,C 180,E1 -2617.31,E2 -2617.31} C_VEL
LIN {X 0,Y 566.14,Z 985,A -85,B 0,C 180,E1 -2618.386,E2 -2618.386} C_VEL
LIN {X 0,Y 566.302,Z 974.614,A -85,B 0,C 180,E1 -2619.463,E2 -2619.463} C_VEL
LIN {X 0,Y 566.421,Z 964.942,A -85,B 0,C 180,E1 -2620.273,E2 -2620.273} C_VEL
LIN {X 0,Y 566.559,Z 954.669,A -85,B 0,C 180,E1 -2620.973,E2 -2620.973} C_VEL
LIN {X 0,Y 566.719,Z 942.908,A -85,B 0,C 180,E1 -2621.606,E2 -2621.606} C_VEL
LIN {X 0,Y 566.813,Z 930.207,A -85,B 0,C 180,E1 -2622.122,E2 -2622.122} C_VEL
LIN {X 0,Y 566.91,Z 917.567,A -85,B 0,C 180,E1 -2622.483,E2 -2622.483} C_VEL
LIN {X 0,Y 567.016,Z 904.402,A -85,B 0,C 180,E1 -2622.708,E2 -2622.708} C_VEL
LIN {X 0,Y 567.103,Z 806.022,A -85,B 0,C 180,E1 -2623.96,E2 -2623.96} C_VEL
LIN {X 0,Y 566.549,Z 801.906,A -85,B 0,C 180,E1 -2624.043,E2 -2624.043} C_VEL
LIN {X 0,Y 566.84,Z 775.456,A -85,B 0,C 180,E1 -2626.919,E2 -2626.919} C_VEL
LIN {X 0,Y 567.209,Z 748.717,A -85,B 0,C 180,E1 -2629.883,E2 -2629.883} C_VEL
LIN {X 0,Y 567.542,Z 724.847,A -85,B 0,C 180,E1 -2632.573,E2 -2632.573} C_VEL
LIN {X 0,Y 567.921,Z 703.583,A -85,B 0,C 180,E1 -2635.008,E2 -2635.008} C_VEL
LIN {X 0,Y 568.14,Z 690.012,A -85,B 0,C 180,E1 -2636.586,E2 -2636.586} C_VEL
LIN {X 0,Y 566.263,Z 682.051,A -85,B 0,C 180,E1 -2637.661,E2 -2637.661} C_VEL
LIN {X 0,Y 566.178,Z 681.96,A -85,B 0,C 180,E1 -2640.591,E2 -2640.591} C_VEL
LIN {X 0,Y 566.201,Z 681.952,A -85,B 0,C 180,E1 -2643.102,E2 -2643.102} C_VEL
LIN {X 0,Y 566.157,Z 681.957,A -85,B 0,C 180,E1 -2645.691,E2 -2645.691} C_VEL
LIN {X 0,Y 566.204,Z 681.96,A -85,B 0,C 180,E1 -2648.557,E2 -2648.557} C_VEL
LIN {X 0,Y 566.167,Z 681.957,A -85,B 0,C 180,E1 -2651.138,E2 -2651.138} C_VEL
LIN {X 0,Y 566.19,Z 681.953,A -85,B 0,C 180,E1 -2654.035,E2 -2654.035} C_VEL
LIN {X 0,Y 566.202,Z 681.957,A -85,B 0,C 180,E1 -2657.081,E2 -2657.081} C_VEL
LIN {X 0,Y 566.219,Z 681.946,A -85,B 0,C 180,E1 -2659.802,E2 -2659.802} C_VEL
LIN {X 0,Y 566.19,Z 681.955,A -85,B 0,C 180,E1 -2662.598,E2 -2662.598} C_VEL
LIN {X 0,Y 566.212,Z 681.957,A -85,B 0,C 180,E1 -2665.182,E2 -2665.182} C_VEL
LIN {X 0,Y 566.222,Z 681.95,A -85,B 0,C 180,E1 -2667.743,E2 -2667.743} C_VEL
LIN {X 0,Y 566.218,Z 681.948,A -85,B 0,C 180,E1 -2670.323,E2 -2670.323} C_VEL
LIN {X 0,Y 566.223,Z 681.957,A -85,B 0,C 180,E1 -2673.335,E2 -2673.335} C_VEL
LIN {X 0,Y 566.188,Z 681.957,A -85,B 0,C 180,E1 -2675.819,E2 -2675.819} C_VEL
LIN {X 0,Y 566.197,Z 681.95,A -85,B 0,C 180,E1 -2678.902,E2 -2678.902} C_VEL
LIN {X 0,Y 566.197,Z 681.953,A -85,B 0,C 180,E1 -2681.172,E2 -2681.172} C_VEL
LIN {X 0,Y 566.201,Z 681.954,A -85,B 0,C 180,E1 -2683.412,E2 -2683.412} C_VEL
LIN {X 0,Y 566.185,Z 681.954,A -85,B 0,C 180,E1 -2686.359,E2 -2686.359} C_VEL
LIN {X 0,Y 566.222,Z 681.948,A -85,B 0,C 180,E1 -2688.675,E2 -2688.675} C_VEL
LIN {X 0,Y 566.217,Z 681.948,A -85,B 0,C 180,E1 -2691.434,E2 -2691.434} C_VEL
LIN {X 0,Y 566.259,Z 681.95,A -85,B 0,C 180,E1 -2694.302,E2 -2694.302} C_VEL
LIN {X 0,Y 566.263,Z 681.946,A -85,B 0,C 180,E1 -2697.866,E2 -2697.866} C_VEL
LIN {X 0,Y 566.298,Z 681.943,A -85,B 0,C 180,E1 -2700.711,E2 -2700.711} C_VEL
LIN {X 0,Y 566.269,Z 681.945,A -85,B 0,C 180,E1 -2702.846,E2 -2702.846} C_VEL
LIN {X 0,Y 566.245,Z 681.944,A -85,B 0,C 180,E1 -2705.699,E2 -2705.699} C_VEL
LIN {X 0,Y 566.222,Z 681.956,A -85,B 0,C 180,E1 -2708.566,E2 -2708.566} C_VEL
LIN {X 0,Y 566.24,Z 681.946,A -85,B 0,C 180,E1 -2711.455,E2 -2711.455} C_VEL
LIN {X 0,Y 566.218,Z 681.953,A -85,B 0,C 180,E1 -2714.505,E2 -2714.505} C_VEL
LIN {X 0,Y 566.186,Z 681.957,A -85,B 0,C 180,E1 -2717.332,E2 -2717.332} C_VEL
LIN {X 0,Y 566.2,Z 681.951,A -85,B 0,C 180,E1 -2720.338,E2 -2720.338} C_VEL
LIN {X 0,Y 566.161,Z 681.962,A -85,B 0,C 180,E1 -2723.282,E2 -2723.282} C_VEL
LIN {X 0,Y 566.195,Z 681.954,A -85,B 0,C 180,E1 -2725.75,E2 -2725.75} C_VEL
LIN {X 0,Y 566.191,Z 681.958,A -85,B 0,C 180,E1 -2727.496,E2 -2727.496} C_VEL
LIN {X 0,Y 565.512,Z 682.037,A -85,B 0,C 180,E1 -2728.09,E2 -2728.09} C_VEL
LIN {X 0,Y 562.647,Z 682.396,A -85,B 0,C 180,E1 -2729.053,E2 -2729.053} C_VEL
LIN {X 0,Y 560.236,Z 682.698,A -85,B 0,C 180,E1 -2729.829,E2 -2729.829} C_VEL
LIN {X 0,Y 559.209,Z 682.822,A -85,B 0,C 180,E1 -2730.428,E2 -2730.428} C_VEL
LIN {X 0,Y 559.129,Z 682.832,A -85,B 0,C 180,E1 -2730.63,E2 -2730.63} C_VEL
LIN {X 0,Y 559.156,Z 682.837,A -85,B 0,C 180,E1 -2733.576,E2 -2733.576} C_VEL
LIN {X 0,Y 559.15,Z 682.829,A -85,B 0,C 180,E1 -2736.448,E2 -2736.448} C_VEL
LIN {X 0,Y 559.166,Z 682.826,A -85,B 0,C 180,E1 -2738.935,E2 -2738.935} C_VEL
LIN {X 0,Y 559.169,Z 682.832,A -85,B 0,C 180,E1 -2742.138,E2 -2742.138} C_VEL
LIN {X 0,Y 559.128,Z 682.833,A -85,B 0,C 180,E1 -2745.262,E2 -2745.262} C_VEL
LIN {X 0,Y 559.154,Z 682.836,A -85,B 0,C 180,E1 -2748.231,E2 -2748.231} C_VEL
LIN {X 0,Y 559.185,Z 682.967,A -85,B 0,C 180,E1 -2751.115,E2 -2751.115} C_VEL
LIN {X 0,Y 559.387,Z 683.946,A -85,B 0,C 180,E1 -2751.237,E2 -2751.237} C_VEL
LIN {X 0,Y 560.245,Z 686.728,A -85,B 0,C 180,E1 -2751.307,E2 -2751.307} C_VEL
LIN {X 0,Y 560.053,Z 762.585,A -85,B 0,C 180,E1 -2752.303,E2 -2752.303} C_VEL
LIN {X 0,Y 559.918,Z 776.336,A -85,B 0,C 180,E1 -2752.643,E2 -2752.643} C_VEL
LIN {X 0,Y 559.781,Z 788.715,A -85,B 0,C 180,E1 -2753.099,E2 -2753.099} C_VEL
LIN {X 0,Y 559.595,Z 801.39,A -85,B 0,C 180,E1 -2753.739,E2 -2753.739} C_VEL
LIN {X 0,Y 559.439,Z 812.79,A -85,B 0,C 180,E1 -2754.479,E2 -2754.479} C_VEL
LIN {X 0,Y 559.28,Z 823.39,A -85,B 0,C 180,E1 -2755.348,E2 -2755.348} C_VEL
LIN {X 0,Y 559.131,Z 832.227,A -85,B 0,C 180,E1 -2756.237,E2 -2756.237} C_VEL
LIN {X 0,Y 559.027,Z 840.687,A -85,B 0,C 180,E1 -2757.278,E2 -2757.278} C_VEL
LIN {X 0,Y 558.956,Z 847.461,A -85,B 0,C 180,E1 -2758.302,E2 -2758.302} C_VEL
LIN {X 0,Y 558.885,Z 853.246,A -85,B 0,C 180,E1 -2759.385,E2 -2759.385} C_VEL
LIN {X 0,Y 558.855,Z 858.379,A -85,B 0,C 180,E1 -2760.631,E2 -2760.631} C_VEL
LIN {X 0,Y 558.788,Z 861.656,A -85,B 0,C 180,E1 -2761.692,E2 -2761.692} C_VEL
LIN {X 0,Y 558.75,Z 864.501,A -85,B 0,C 180,E1 -2763.077,E2 -2763.077} C_VEL
LIN {X 0,Y 558.734,Z 865.485,A -85,B 0,C 180,E1 -2763.882,E2 -2763.882} C_VEL
LIN {X 0,Y 558.742,Z 865.977,A -85,B 0,C 180,E1 -2764.91,E2 -2764.91} C_VEL
LIN {X 0,Y 558.73,Z 865.424,A -85,B 0,C 180,E1 -2766.266,E2 -2766.266} C_VEL
LIN {X 0,Y 558.734,Z 864.437,A -85,B 0,C 180,E1 -2767.051,E2 -2767.051} C_VEL
LIN {X 0,Y 558.755,Z 863.008,A -85,B 0,C 180,E1 -2767.832,E2 -2767.832} C_VEL
LIN {X 0,Y 558.832,Z 859.934,A -85,B 0,C 180,E1 -2768.998,E2 -2768.998} C_VEL
LIN {X 0,Y 558.881,Z 855.713,A -85,B 0,C 180,E1 -2770.153,E2 -2770.153} C_VEL
LIN {X 0,Y 558.922,Z 849.165,A -85,B 0,C 180,E1 -2771.49,E2 -2771.49} C_VEL
LIN {X 0,Y 558.994,Z 841.584,A -85,B 0,C 180,E1 -2772.691,E2 -2772.691} C_VEL
LIN {X 0,Y 559.139,Z 833.049,A -85,B 0,C 180,E1 -2773.761,E2 -2773.761} C_VEL
LIN {X 0,Y 559.237,Z 822.764,A -85,B 0,C 180,E1 -2774.802,E2 -2774.802} C_VEL
LIN {X 0,Y 559.398,Z 812.467,A -85,B 0,C 180,E1 -2775.634,E2 -2775.634} C_VEL
LIN {X 0,Y 559.614,Z 800.857,A -85,B 0,C 180,E1 -2776.382,E2 -2776.382} C_VEL
LIN {X 0,Y 559.776,Z 788.823,A -85,B 0,C 180,E1 -2776.986,E2 -2776.986} C_VEL
LIN {X 0,Y 559.898,Z 776.25,A -85,B 0,C 180,E1 -2777.45,E2 -2777.45} C_VEL
LIN {X 0,Y 560.037,Z 763.265,A -85,B 0,C 180,E1 -2777.774,E2 -2777.774} C_VEL
LIN {X 0,Y 560.169,Z 725.199,A -85,B 0,C 180,E1 -2778.288,E2 -2778.288} C_VEL
LIN {X 0,Y 560.058,Z 686.026,A -85,B 0,C 180,E1 -2778.796,E2 -2778.796} C_VEL
LIN {X 0,Y 559.32,Z 683.606,A -85,B 0,C 180,E1 -2778.876,E2 -2778.876} C_VEL
LIN {X 0,Y 559.177,Z 682.861,A -85,B 0,C 180,E1 -2779.039,E2 -2779.039} C_VEL
LIN {X 0,Y 559.144,Z 682.84,A -85,B 0,C 180,E1 -2782.054,E2 -2782.054} C_VEL
LIN {X 0,Y 559.229,Z 682.82,A -85,B 0,C 180,E1 -2784.954,E2 -2784.954} C_VEL
LIN {X 0,Y 559.25,Z 682.822,A -85,B 0,C 180,E1 -2787.84,E2 -2787.84} C_VEL
LIN {X 0,Y 559.257,Z 682.823,A -85,B 0,C 180,E1 -2790.001,E2 -2790.001} C_VEL
LIN {X 0,Y 559.212,Z 682.824,A -85,B 0,C 180,E1 -2792.883,E2 -2792.883} C_VEL
LIN {X 0,Y 559.199,Z 682.824,A -85,B 0,C 180,E1 -2795.772,E2 -2795.772} C_VEL
LIN {X 0,Y 559.155,Z 682.836,A -85,B 0,C 180,E1 -2798.676,E2 -2798.676} C_VEL
LIN {X 0,Y 559.136,Z 682.83,A -85,B 0,C 180,E1 -2801.603,E2 -2801.603} C_VEL
LIN {X 0,Y 559.166,Z 682.835,A -85,B 0,C 180,E1 -2804.58,E2 -2804.58} C_VEL
LIN {X 0,Y 559.125,Z 682.832,A -85,B 0,C 180,E1 -2807.559,E2 -2807.559} C_VEL
LIN {X 0,Y 559.153,Z 682.831,A -85,B 0,C 180,E1 -2810.607,E2 -2810.607} C_VEL
LIN {X 0,Y 559.136,Z 682.833,A -85,B 0,C 180,E1 -2813.426,E2 -2813.426} C_VEL
LIN {X 0,Y 559.116,Z 682.83,A -85,B 0,C 180,E1 -2816.101,E2 -2816.101} C_VEL
LIN {X 0,Y 559.103,Z 682.835,A -85,B 0,C 180,E1 -2818.534,E2 -2818.534} C_VEL
LIN {X 0,Y 559.12,Z 682.841,A -85,B 0,C 180,E1 -2821.268,E2 -2821.268} C_VEL
LIN {X 0,Y 559.13,Z 682.828,A -85,B 0,C 180,E1 -2823.943,E2 -2823.943} C_VEL
LIN {X 0,Y 559.102,Z 682.832,A -85,B 0,C 180,E1 -2826.438,E2 -2826.438} C_VEL
LIN {X 0,Y 559.111,Z 682.836,A -85,B 0,C 180,E1 -2828.94,E2 -2828.94} C_VEL
LIN {X 0,Y 559.094,Z 682.842,A -85,B 0,C 180,E1 -2831.778,E2 -2831.778} C_VEL
LIN {X 0,Y 559.121,Z 682.832,A -85,B 0,C 180,E1 -2834.742,E2 -2834.742} C_VEL
LIN {X 0,Y 559.114,Z 682.841,A -85,B 0,C 180,E1 -2837.871,E2 -2837.871} C_VEL
LIN {X 0,Y 559.145,Z 682.834,A -85,B 0,C 180,E1 -2840.131,E2 -2840.131} C_VEL
LIN {X 0,Y 559.071,Z 682.839,A -85,B 0,C 180,E1 -2842.886,E2 -2842.886} C_VEL
LIN {X 0,Y 559.121,Z 682.837,A -85,B 0,C 180,E1 -2845.553,E2 -2845.553} C_VEL
LIN {X 0,Y 559.137,Z 682.84,A -85,B 0,C 180,E1 -2848.135,E2 -2848.135} C_VEL
LIN {X 0,Y 559.095,Z 682.841,A -85,B 0,C 180,E1 -2850.643,E2 -2850.643} C_VEL
LIN {X 0,Y 559.143,Z 683.045,A -85,B 0,C 180,E1 -2853.132,E2 -2853.132} C_VEL
LIN {X 0,Y 559.355,Z 683.93,A -85,B 0,C 180,E1 -2853.236,E2 -2853.236} C_VEL
LIN {X 0,Y 560.204,Z 686.633,A -85,B 0,C 180,E1 -2853.305,E2 -2853.305} C_VEL
LIN {X 0,Y 560.03,Z 761.745,A -85,B 0,C 180,E1 -2854.289,E2 -2854.289} C_VEL
LIN {X 0,Y 559.923,Z 773.996,A -85,B 0,C 180,E1 -2854.577,E2 -2854.577} C_VEL
LIN {X 0,Y 559.815,Z 784.483,A -85,B 0,C 180,E1 -2854.931,E2 -2854.931} C_VEL
LIN {X 0,Y 559.635,Z 795.389,A -85,B 0,C 180,E1 -2855.418,E2 -2855.418} C_VEL
LIN {X 0,Y 559.533,Z 804.184,A -85,B 0,C 180,E1 -2855.907,E2 -2855.907} C_VEL
LIN {X 0,Y 559.394,Z 814.262,A -85,B 0,C 180,E1 -2856.595,E2 -2856.595} C_VEL
LIN {X 0,Y 559.247,Z 823.512,A -85,B 0,C 180,E1 -2857.365,E2 -2857.365} C_VEL
LIN {X 0,Y 559.149,Z 831.797,A -85,B 0,C 180,E1 -2858.198,E2 -2858.198} C_VEL
LIN {X 0,Y 559.027,Z 838.581,A -85,B 0,C 180,E1 -2859.004,E2 -2859.004} C_VEL
LIN {X 0,Y 558.955,Z 845.311,A -85,B 0,C 180,E1 -2859.963,E2 -2859.963} C_VEL
LIN {X 0,Y 558.904,Z 850.843,A -85,B 0,C 180,E1 -2860.917,E2 -2860.917} C_VEL
LIN {X 0,Y 558.828,Z 856.136,A -85,B 0,C 180,E1 -2862.054,E2 -2862.054} C_VEL
LIN {X 0,Y 558.819,Z 860.175,A -85,B 0,C 180,E1 -2863.186,E2 -2863.186} C_VEL
LIN {X 0,Y 558.754,Z 862.257,A -85,B 0,C 180,E1 -2863.936,E2 -2863.936} C_VEL
LIN {X 0,Y 558.721,Z 863.856,A -85,B 0,C 180,E1 -2864.683,E2 -2864.683} C_VEL
LIN {X 0,Y 558.764,Z 865.147,A -85,B 0,C 180,E1 -2865.58,E2 -2865.58} C_VEL
LIN {X 0,Y 558.745,Z 865.978,A -85,B 0,C 180,E1 -2866.914,E2 -2866.914} C_VEL
LIN {X 0,Y 558.778,Z 865.288,A -85,B 0,C 180,E1 -2868.39,E2 -2868.39} C_VEL
LIN {X 0,Y 558.796,Z 864.327,A -85,B 0,C 180,E1 -2869.125,E2 -2869.125} C_VEL
LIN {X 0,Y 558.778,Z 861.13,A -85,B 0,C 180,E1 -2870.589,E2 -2870.589} C_VEL
LIN {X 0,Y 558.83,Z 857.555,A -85,B 0,C 180,E1 -2871.684,E2 -2871.684} C_VEL
LIN {X 0,Y 558.891,Z 852.875,A -85,B 0,C 180,E1 -2872.776,E2 -2872.776} C_VEL
LIN {X 0,Y 558.927,Z 846.965,A -85,B 0,C 180,E1 -2873.864,E2 -2873.864} C_VEL
LIN {X 0,Y 558.951,Z 840.981,A -85,B 0,C 180,E1 -2874.77,E2 -2874.77} C_VEL
LIN {X 0,Y 559.122,Z 833.772,A -85,B 0,C 180,E1 -2875.675,E2 -2875.675} C_VEL
LIN {X 0,Y 559.209,Z 825.114,A -85,B 0,C 180,E1 -2876.577,E2 -2876.577} C_VEL
LIN {X 0,Y 559.356,Z 816.796,A -85,B 0,C 180,E1 -2877.299,E2 -2877.299} C_VEL
LIN {X 0,Y 559.498,Z 808.134,A -85,B 0,C 180,E1 -2877.93,E2 -2877.93} C_VEL
LIN {X 0,Y 559.581,Z 797.545,A -85,B 0,C 180,E1 -2878.561,E2 -2878.561} C_VEL
LIN {X 0,Y 559.796,Z 787.001,A -85,B 0,C 180,E1 -2879.056,E2 -2879.056} C_VEL
LIN {X 0,Y 559.914,Z 776.451,A -85,B 0,C 180,E1 -2879.438,E2 -2879.438} C_VEL
LIN {X 0,Y 559.979,Z 765.234,A -85,B 0,C 180,E1 -2879.73,E2 -2879.73} C_VEL
LIN {X 0,Y 560.105,Z 751.123,A -85,B 0,C 180,E1 -2879.955,E2 -2879.955} C_VEL
LIN {X 0,Y 560.169,Z 686.169,A -85,B 0,C 180,E1 -2880.792,E2 -2880.792} C_VEL
LIN {X 0,Y 559.358,Z 683.553,A -85,B 0,C 180,E1 -2880.877,E2 -2880.877} C_VEL
LIN {X 0,Y 559.224,Z 682.868,A -85,B 0,C 180,E1 -2881.035,E2 -2881.035} C_VEL
LIN {X 0,Y 559.238,Z 682.822,A -85,B 0,C 180,E1 -2882.881,E2 -2882.881} C_VEL
LIN {X 0,Y 559.226,Z 682.827,A -85,B 0,C 180,E1 -2885.77,E2 -2885.77} C_VEL
LIN {X 0,Y 559.174,Z 682.829,A -85,B 0,C 180,E1 -2888.675,E2 -2888.675} C_VEL
LIN {X 0,Y 559.212,Z 682.823,A -85,B 0,C 180,E1 -2891.6,E2 -2891.6} C_VEL
LIN {X 0,Y 559.208,Z 682.828,A -85,B 0,C 180,E1 -2894.595,E2 -2894.595} C_VEL
LIN {X 0,Y 559.144,Z 682.83,A -85,B 0,C 180,E1 -2897.557,E2 -2897.557} C_VEL
LIN {X 0,Y 559.172,Z 682.828,A -85,B 0,C 180,E1 -2899.837,E2 -2899.837} C_VEL
LIN {X 0,Y 559.146,Z 682.833,A -85,B 0,C 180,E1 -2902.153,E2 -2902.153} C_VEL
LIN {X 0,Y 559.181,Z 682.827,A -85,B 0,C 180,E1 -2905.298,E2 -2905.298} C_VEL
LIN {X 0,Y 559.134,Z 682.831,A -85,B 0,C 180,E1 -2907.715,E2 -2907.715} C_VEL
LIN {X 0,Y 559.159,Z 682.829,A -85,B 0,C 180,E1 -2910.182,E2 -2910.182} C_VEL
LIN {X 0,Y 559.157,Z 682.835,A -85,B 0,C 180,E1 -2912.715,E2 -2912.715} C_VEL
LIN {X 0,Y 559.133,Z 682.836,A -85,B 0,C 180,E1 -2915.324,E2 -2915.324} C_VEL
LIN {X 0,Y 559.137,Z 682.831,A -85,B 0,C 180,E1 -2918.017,E2 -2918.017} C_VEL
LIN {X 0,Y 559.161,Z 682.832,A -85,B 0,C 180,E1 -2920.812,E2 -2920.812} C_VEL
LIN {X 0,Y 559.144,Z 682.833,A -85,B 0,C 180,E1 -2923.734,E2 -2923.734} C_VEL
LIN {X 0,Y 559.151,Z 682.831,A -85,B 0,C 180,E1 -2926.803,E2 -2926.803} C_VEL
LIN {X 0,Y 559.161,Z 682.834,A -85,B 0,C 180,E1 -2929.187,E2 -2929.187} C_VEL
LIN {X 0,Y 559.135,Z 682.834,A -85,B 0,C 180,E1 -2931.982,E2 -2931.982} C_VEL
LIN {X 0,Y 559.134,Z 682.832,A -85,B 0,C 180,E1 -2934.787,E2 -2934.787} C_VEL
LIN {X 0,Y 559.159,Z 682.834,A -85,B 0,C 180,E1 -2937.364,E2 -2937.364} C_VEL
LIN {X 0,Y 559.153,Z 682.837,A -85,B 0,C 180,E1 -2940.142,E2 -2940.142} C_VEL
LIN {X 0,Y 559.195,Z 683.037,A -85,B 0,C 180,E1 -2942.188,E2 -2942.188} C_VEL
LIN {X 0,Y 561.233,Z 691.107,A -85,B 0,C 180,E1 -2943.204,E2 -2943.204} C_VEL
LIN {X 0,Y 561.354,Z 697.931,A -85,B 0,C 180,E1 -2944.011,E2 -2944.011} C_VEL
LIN {X 0,Y 560.755,Z 724.827,A -85,B 0,C 180,E1 -2947.136,E2 -2947.136} C_VEL
LIN {X 0,Y 560.343,Z 748.697,A -85,B 0,C 180,E1 -2949.861,E2 -2949.861} C_VEL
LIN {X 0,Y 559.925,Z 775.791,A -85,B 0,C 180,E1 -2952.903,E2 -2952.903} C_VEL
LIN {X 0,Y 559.571,Z 801.875,A -85,B 0,C 180,E1 -2955.776,E2 -2955.776} C_VEL
LIN {X 0,Y 560.319,Z 809.431,A -85,B 0,C 180,E1 -2955.911,E2 -2955.911} C_VEL
LIN {X 0,Y 560.031,Z 911.896,A -85,B 0,C 180,E1 -2957.244,E2 -2957.244} C_VEL
LIN {X 0,Y 559.98,Z 924.424,A -85,B 0,C 180,E1 -2957.542,E2 -2957.542} C_VEL
LIN {X 0,Y 559.793,Z 936.893,A -85,B 0,C 180,E1 -2957.979,E2 -2957.979} C_VEL
LIN {X 0,Y 559.671,Z 948.788,A -85,B 0,C 180,E1 -2958.546,E2 -2958.546} C_VEL
LIN {X 0,Y 559.505,Z 959.896,A -85,B 0,C 180,E1 -2959.23,E2 -2959.23} C_VEL
LIN {X 0,Y 559.309,Z 970.529,A -85,B 0,C 180,E1 -2960.05,E2 -2960.05} C_VEL
LIN {X 0,Y 559.162,Z 980.055,A -85,B 0,C 180,E1 -2960.96,E2 -2960.96} C_VEL
LIN {X 0,Y 559.048,Z 987.952,A -85,B 0,C 180,E1 -2961.868,E2 -2961.868} C_VEL
LIN {X 0,Y 558.945,Z 995.615,A -85,B 0,C 180,E1 -2962.957,E2 -2962.957} C_VEL
LIN {X 0,Y 558.936,Z 1002.675,A -85,B 0,C 180,E1 -2964.226,E2 -2964.226} C_VEL
LIN {X 0,Y 558.826,Z 1007.368,A -85,B 0,C 180,E1 -2965.31,E2 -2965.31} C_VEL
LIN {X 0,Y 558.836,Z 1010.954,A -85,B 0,C 180,E1 -2966.394,E2 -2966.394} C_VEL
LIN {X 0,Y 558.799,Z 1012.806,A -85,B 0,C 180,E1 -2967.115,E2 -2967.115} C_VEL
LIN {X 0,Y 558.745,Z 1015.185,A -85,B 0,C 180,E1 -2968.557,E2 -2968.557} C_VEL
LIN {X 0,Y 558.74,Z 1016,A -85,B 0,C 180,E1 -2969.999,E2 -2969.999} C_VEL
LIN {X 0,Y 558.745,Z 1015.188,A -85,B 0,C 180,E1 -2971.44,E2 -2971.44} C_VEL
LIN {X 0,Y 558.799,Z 1012.812,A -85,B 0,C 180,E1 -2972.883,E2 -2972.883} C_VEL
LIN {X 0,Y 558.843,Z 1009.899,A -85,B 0,C 180,E1 -2973.965,E2 -2973.965} C_VEL
LIN {X 0,Y 558.798,Z 1005.953,A -85,B 0,C 180,E1 -2975.05,E2 -2975.05} C_VEL
LIN {X 0,Y 558.925,Z 1000.872,A -85,B 0,C 180,E1 -2976.134,E2 -2976.134} C_VEL
LIN {X 0,Y 558.976,Z 994.476,A -85,B 0,C 180,E1 -2977.222,E2 -2977.222} C_VEL
LIN {X 0,Y 559.09,Z 986.488,A -85,B 0,C 180,E1 -2978.311,E2 -2978.311} C_VEL
LIN {X 0,Y 559.236,Z 976.55,A -85,B 0,C 180,E1 -2979.402,E2 -2979.402} C_VEL
LIN {X 0,Y 559.41,Z 966.113,A -85,B 0,C 180,E1 -2980.312,E2 -2980.312} C_VEL
LIN {X 0,Y 559.564,Z 954.912,A -85,B 0,C 180,E1 -2981.097,E2 -2981.097} C_VEL
LIN {X 0,Y 559.758,Z 942.909,A -85,B 0,C 180,E1 -2981.753,E2 -2981.753} C_VEL
LIN {X 0,Y 559.887,Z 930.206,A -85,B 0,C 180,E1 -2982.274,E2 -2982.274} C_VEL
LIN {X 0,Y 559.977,Z 917.566,A -85,B 0,C 180,E1 -2982.64,E2 -2982.64} C_VEL
LIN {X 0,Y 560.111,Z 904.402,A -85,B 0,C 180,E1 -2982.868,E2 -2982.868} C_VEL
LIN {X 0,Y 560.163,Z 806.372,A -85,B 0,C 180,E1 -2984.132,E2 -2984.132} C_VEL
LIN {X 0,Y 559.574,Z 801.911,A -85,B 0,C 180,E1 -2984.222,E2 -2984.222} C_VEL
LIN {X 0,Y 559.922,Z 774.771,A -85,B 0,C 180,E1 -2987.211,E2 -2987.211} C_VEL
LIN {X 0,Y 560.335,Z 748.385,A -85,B 0,C 180,E1 -2990.175,E2 -2990.175} C_VEL
LIN {X 0,Y 560.752,Z 724.847,A -85,B 0,C 180,E1 -2992.862,E2 -2992.862} C_VEL
LIN {X 0,Y 561.28,Z 700.924,A -85,B 0,C 180,E1 -2995.638,E2 -2995.638} C_VEL
LIN {X 0,Y 561.45,Z 692.892,A -85,B 0,C 180,E1 -2996.582,E2 -2996.582} C_VEL
LIN {X 0,Y 559.227,Z 682.923,A -85,B 0,C 180,E1 -2997.834,E2 -2997.834} C_VEL
LIN {X 0,Y 559.152,Z 682.831,A -85,B 0,C 180,E1 -3001.018,E2 -3001.018} C_VEL
LIN {X 0,Y 559.16,Z 682.832,A -85,B 0,C 180,E1 -3003.948,E2 -3003.948} C_VEL
LIN {X 0,Y 559.135,Z 682.833,A -85,B 0,C 180,E1 -3007.107,E2 -3007.107} C_VEL
LIN {X 0,Y 559.154,Z 682.83,A -85,B 0,C 180,E1 -3009.941,E2 -3009.941} C_VEL
LIN {X 0,Y 559.151,Z 682.837,A -85,B 0,C 180,E1 -3012.743,E2 -3012.743} C_VEL
LIN {X 0,Y 559.148,Z 682.828,A -85,B 0,C 180,E1 -3015.759,E2 -3015.759} C_VEL
LIN {X 0,Y 559.184,Z 682.826,A -85,B 0,C 180,E1 -3018.232,E2 -3018.232} C_VEL
LIN {X 0,Y 559.17,Z 682.833,A -85,B 0,C 180,E1 -3021.19,E2 -3021.19} C_VEL
LIN {X 0,Y 559.164,Z 682.826,A -85,B 0,C 180,E1 -3023.791,E2 -3023.791} C_VEL
LIN {X 0,Y 559.155,Z 682.828,A -85,B 0,C 180,E1 -3026.425,E2 -3026.425} C_VEL
LIN {X 0,Y 559.149,Z 682.835,A -85,B 0,C 180,E1 -3028.98,E2 -3028.98} C_VEL
LIN {X 0,Y 559.161,Z 682.833,A -85,B 0,C 180,E1 -3031.617,E2 -3031.617} C_VEL
LIN {X 0,Y 559.188,Z 682.827,A -85,B 0,C 180,E1 -3033.903,E2 -3033.903} C_VEL
LIN {X 0,Y 559.146,Z 682.829,A -85,B 0,C 180,E1 -3036.567,E2 -3036.567} C_VEL
LIN {X 0,Y 559.169,Z 682.832,A -85,B 0,C 180,E1 -3039.395,E2 -3039.395} C_VEL
LIN {X 0,Y 559.14,Z 682.84,A -85,B 0,C 180,E1 -3041.686,E2 -3041.686} C_VEL
LIN {X 0,Y 559.153,Z 682.836,A -85,B 0,C 180,E1 -3043.948,E2 -3043.948} C_VEL
LIN {X 0,Y 559.16,Z 682.831,A -85,B 0,C 180,E1 -3046.184,E2 -3046.184} C_VEL
LIN {X 0,Y 559.193,Z 682.824,A -85,B 0,C 180,E1 -3048.604,E2 -3048.604} C_VEL
LIN {X 0,Y 559.176,Z 682.824,A -85,B 0,C 180,E1 -3051.326,E2 -3051.326} C_VEL
LIN {X 0,Y 559.226,Z 682.828,A -85,B 0,C 180,E1 -3054.23,E2 -3054.23} C_VEL
LIN {X 0,Y 559.235,Z 682.821,A -85,B 0,C 180,E1 -3057.839,E2 -3057.839} C_VEL
LIN {X 0,Y 559.267,Z 682.818,A -85,B 0,C 180,E1 -3060.72,E2 -3060.72} C_VEL
LIN {X 0,Y 559.234,Z 682.821,A -85,B 0,C 180,E1 -3062.882,E2 -3062.882} C_VEL
LIN {X 0,Y 559.214,Z 682.82,A -85,B 0,C 180,E1 -3065.77,E2 -3065.77} C_VEL
LIN {X 0,Y 559.181,Z 682.834,A -85,B 0,C 180,E1 -3068.675,E2 -3068.675} C_VEL
LIN {X 0,Y 559.198,Z 682.822,A -85,B 0,C 180,E1 -3071.601,E2 -3071.601} C_VEL
LIN {X 0,Y 559.188,Z 682.83,A -85,B 0,C 180,E1 -3074.596,E2 -3074.596} C_VEL
LIN {X 0,Y 559.13,Z 682.833,A -85,B 0,C 180,E1 -3077.558,E2 -3077.558} C_VEL
LIN {X 0,Y 559.16,Z 682.828,A -85,B 0,C 180,E1 -3079.838,E2 -3079.838} C_VEL
LIN {X 0,Y 559.129,Z 682.83,A -85,B 0,C 180,E1 -3082.154,E2 -3082.154} C_VEL
LIN {X 0,Y 559.141,Z 682.837,A -85,B 0,C 180,E1 -3085.182,E2 -3085.182} C_VEL
LIN {X 0,Y 559.146,Z 682.831,A -85,B 0,C 180,E1 -3087.714,E2 -3087.714} C_VEL
LIN {X 0,Y 559.129,Z 682.832,A -85,B 0,C 180,E1 -3090.63,E2 -3090.63} C_VEL
LIN {X 0,Y 558.47,Z 682.923,A -85,B 0,C 180,E1 -3091.232,E2 -3091.232} C_VEL
LIN {X 0,Y 555.61,Z 683.271,A -85,B 0,C 180,E1 -3092.208,E2 -3092.208} C_VEL
LIN {X 0,Y 553.199,Z 683.571,A -85,B 0,C 180,E1 -3092.994,E2 -3092.994} C_VEL
LIN {X 0,Y 552.179,Z 683.706,A -85,B 0,C 180,E1 -3093.601,E2 -3093.601} C_VEL
LIN {X 0,Y 552.104,Z 683.708,A -85,B 0,C 180,E1 -3093.806,E2 -3093.806} C_VEL
LIN {X 0,Y 552.1,Z 683.707,A -85,B 0,C 180,E1 -3096.748,E2 -3096.748} C_VEL
LIN {X 0,Y 552.121,Z 683.71,A -85,B 0,C 180,E1 -3099.528,E2 -3099.528} C_VEL
LIN {X 0,Y 552.124,Z 683.706,A -85,B 0,C 180,E1 -3102.427,E2 -3102.427} C_VEL
LIN {X 0,Y 552.087,Z 683.714,A -85,B 0,C 180,E1 -3105.563,E2 -3105.563} C_VEL
LIN {X 0,Y 552.114,Z 683.708,A -85,B 0,C 180,E1 -3108.68,E2 -3108.68} C_VEL
LIN {X 0,Y 552.153,Z 683.926,A -85,B 0,C 180,E1 -3110.955,E2 -3110.955} C_VEL
LIN {X 0,Y 552.381,Z 684.955,A -85,B 0,C 180,E1 -3111.063,E2 -3111.063} C_VEL
LIN {X 0,Y 553.3,Z 687.766,A -85,B 0,C 180,E1 -3111.134,E2 -3111.134} C_VEL
LIN {X 0,Y 553.146,Z 762.91,A -85,B 0,C 180,E1 -3112.136,E2 -3112.136} C_VEL
LIN {X 0,Y 552.992,Z 776.303,A -85,B 0,C 180,E1 -3112.467,E2 -3112.467} C_VEL
LIN {X 0,Y 552.859,Z 788.434,A -85,B 0,C 180,E1 -3112.915,E2 -3112.915} C_VEL
LIN {X 0,Y 552.676,Z 800.556,A -85,B 0,C 180,E1 -3113.526,E2 -3113.526} C_VEL
LIN {X 0,Y 552.495,Z 812.222,A -85,B 0,C 180,E1 -3114.29,E2 -3114.29} C_VEL
LIN {X 0,Y 552.273,Z 821.739,A -85,B 0,C 180,E1 -3115.066,E2 -3115.066} C_VEL
LIN {X 0,Y 552.119,Z 830.593,A -85,B 0,C 180,E1 -3115.94,E2 -3115.94} C_VEL
LIN {X 0,Y 551.924,Z 839.536,A -85,B 0,C 180,E1 -3117.021,E2 -3117.021} C_VEL
LIN {X 0,Y 551.887,Z 846.751,A -85,B 0,C 180,E1 -3118.099,E2 -3118.099} C_VEL
LIN {X 0,Y 551.795,Z 851.57,A -85,B 0,C 180,E1 -3118.972,E2 -3118.972} C_VEL
LIN {X 0,Y 551.729,Z 857.056,A -85,B 0,C 180,E1 -3120.214,E2 -3120.214} C_VEL
LIN {X 0,Y 551.704,Z 861.325,A -85,B 0,C 180,E1 -3121.519,E2 -3121.519} C_VEL
LIN {X 0,Y 551.652,Z 864.575,A -85,B 0,C 180,E1 -3123.101,E2 -3123.101} C_VEL
LIN {X 0,Y 551.626,Z 865.797,A -85,B 0,C 180,E1 -3124.332,E2 -3124.332} C_VEL
LIN {X 0,Y 551.639,Z 865.986,A -85,B 0,C 180,E1 -3125.14,E2 -3125.14} C_VEL
LIN {X 0,Y 551.655,Z 865.151,A -85,B 0,C 180,E1 -3126.531,E2 -3126.531} C_VEL
LIN {X 0,Y 551.653,Z 863.675,A -85,B 0,C 180,E1 -3127.532,E2 -3127.532} C_VEL
LIN {X 0,Y 551.693,Z 861.689,A -85,B 0,C 180,E1 -3128.427,E2 -3128.427} C_VEL
LIN {X 0,Y 551.745,Z 858.446,A -85,B 0,C 180,E1 -3129.496,E2 -3129.496} C_VEL
LIN {X 0,Y 551.838,Z 853.759,A -85,B 0,C 180,E1 -3130.664,E2 -3130.664} C_VEL
LIN {X 0,Y 551.873,Z 847.783,A -85,B 0,C 180,E1 -3131.821,E2 -3131.821} C_VEL
LIN {X 0,Y 551.941,Z 840.251,A -85,B 0,C 180,E1 -3132.972,E2 -3132.972} C_VEL
LIN {X 0,Y 552.12,Z 830.881,A -85,B 0,C 180,E1 -3134.118,E2 -3134.118} C_VEL
LIN {X 0,Y 552.304,Z 820.133,A -85,B 0,C 180,E1 -3135.163,E2 -3135.163} C_VEL
LIN {X 0,Y 552.509,Z 809.247,A -85,B 0,C 180,E1 -3136.015,E2 -3136.015} C_VEL
LIN {X 0,Y 552.686,Z 798.584,A -85,B 0,C 180,E1 -3136.676,E2 -3136.676} C_VEL
LIN {X 0,Y 552.906,Z 786.757,A -85,B 0,C 180,E1 -3137.242,E2 -3137.242} C_VEL
LIN {X 0,Y 553.042,Z 773.932,A -85,B 0,C 180,E1 -3137.693,E2 -3137.693} C_VEL
LIN {X 0,Y 553.174,Z 760.765,A -85,B 0,C 180,E1 -3137.99,E2 -3137.99} C_VEL
LIN {X 0,Y 553.282,Z 687.65,A -85,B 0,C 180,E1 -3138.957,E2 -3138.957} C_VEL
LIN {X 0,Y 552.321,Z 684.627,A -85,B 0,C 180,E1 -3139.044,E2 -3139.044} C_VEL
LIN {X 0,Y 552.141,Z 683.743,A -85,B 0,C 180,E1 -3139.203,E2 -3139.203} C_VEL
LIN {X 0,Y 552.113,Z 683.714,A -85,B 0,C 180,E1 -3141.952,E2 -3141.952} C_VEL
LIN {X 0,Y 552.206,Z 683.695,A -85,B 0,C 180,E1 -3144.89,E2 -3144.89} C_VEL
LIN {X 0,Y 552.221,Z 683.698,A -85,B 0,C 180,E1 -3147.813,E2 -3147.813} C_VEL
LIN {X 0,Y 552.225,Z 683.699,A -85,B 0,C 180,E1 -3150.001,E2 -3150.001} C_VEL
LIN {X 0,Y 552.179,Z 683.7,A -85,B 0,C 180,E1 -3152.919,E2 -3152.919} C_VEL
LIN {X 0,Y 552.171,Z 683.701,A -85,B 0,C 180,E1 -3155.845,E2 -3155.845} C_VEL
LIN {X 0,Y 552.128,Z 683.709,A -85,B 0,C 180,E1 -3158.787,E2 -3158.787} C_VEL
LIN {X 0,Y 552.085,Z 683.709,A -85,B 0,C 180,E1 -3161.753,E2 -3161.753} C_VEL
LIN {X 0,Y 552.128,Z 683.711,A -85,B 0,C 180,E1 -3164.75,E2 -3164.75} C_VEL
LIN {X 0,Y 552.085,Z 683.709,A -85,B 0,C 180,E1 -3167.79,E2 -3167.79} C_VEL
LIN {X 0,Y 552.109,Z 683.703,A -85,B 0,C 180,E1 -3170.103,E2 -3170.103} C_VEL
LIN {X 0,Y 552.084,Z 683.711,A -85,B 0,C 180,E1 -3172.452,E2 -3172.452} C_VEL
LIN {X 0,Y 552.066,Z 683.713,A -85,B 0,C 180,E1 -3175.329,E2 -3175.329} C_VEL
LIN {X 0,Y 552.053,Z 683.711,A -85,B 0,C 180,E1 -3178.102,E2 -3178.102} C_VEL
LIN {X 0,Y 552.068,Z 683.713,A -85,B 0,C 180,E1 -3180.612,E2 -3180.612} C_VEL
LIN {X 0,Y 552.083,Z 683.717,A -85,B 0,C 180,E1 -3183.189,E2 -3183.189} C_VEL
LIN {X 0,Y 552.067,Z 683.71,A -85,B 0,C 180,E1 -3185.846,E2 -3185.846} C_VEL
LIN {X 0,Y 552.065,Z 683.711,A -85,B 0,C 180,E1 -3188.594,E2 -3188.594} C_VEL
LIN {X 0,Y 552.055,Z 683.722,A -85,B 0,C 180,E1 -3191.453,E2 -3191.453} C_VEL
LIN {X 0,Y 552.069,Z 683.711,A -85,B 0,C 180,E1 -3194.528,E2 -3194.528} C_VEL
LIN {X 0,Y 552.085,Z 683.717,A -85,B 0,C 180,E1 -3197.591,E2 -3197.591} C_VEL
LIN {X 0,Y 552.074,Z 683.711,A -85,B 0,C 180,E1 -3200.946,E2 -3200.946} C_VEL
LIN {X 0,Y 552.051,Z 683.72,A -85,B 0,C 180,E1 -3204.153,E2 -3204.153} C_VEL
LIN {X 0,Y 552.099,Z 683.708,A -85,B 0,C 180,E1 -3207.158,E2 -3207.158} C_VEL
LIN {X 0,Y 552.079,Z 683.719,A -85,B 0,C 180,E1 -3209.958,E2 -3209.958} C_VEL
LIN {X 0,Y 552.103,Z 683.886,A -85,B 0,C 180,E1 -3212.953,E2 -3212.953} C_VEL
LIN {X 0,Y 552.287,Z 684.794,A -85,B 0,C 180,E1 -3213.067,E2 -3213.067} C_VEL
LIN {X 0,Y 553.351,Z 688.631,A -85,B 0,C 180,E1 -3213.158,E2 -3213.158} C_VEL
LIN {X 0,Y 553.114,Z 761.738,A -85,B 0,C 180,E1 -3214.127,E2 -3214.127} C_VEL
LIN {X 0,Y 552.994,Z 774.124,A -85,B 0,C 180,E1 -3214.423,E2 -3214.423} C_VEL
LIN {X 0,Y 552.849,Z 785.164,A -85,B 0,C 180,E1 -3214.805,E2 -3214.805} C_VEL
LIN {X 0,Y 552.744,Z 793.864,A -85,B 0,C 180,E1 -3215.191,E2 -3215.191} C_VEL
LIN {X 0,Y 552.546,Z 804.451,A -85,B 0,C 180,E1 -3215.782,E2 -3215.782} C_VEL
LIN {X 0,Y 552.421,Z 813.94,A -85,B 0,C 180,E1 -3216.437,E2 -3216.437} C_VEL
LIN {X 0,Y 552.21,Z 822.635,A -85,B 0,C 180,E1 -3217.159,E2 -3217.159} C_VEL
LIN {X 0,Y 552.099,Z 830.534,A -85,B 0,C 180,E1 -3217.943,E2 -3217.943} C_VEL
LIN {X 0,Y 552.019,Z 837.25,A -85,B 0,C 180,E1 -3218.725,E2 -3218.725} C_VEL
LIN {X 0,Y 551.872,Z 844.201,A -85,B 0,C 180,E1 -3219.694,E2 -3219.694} C_VEL
LIN {X 0,Y 551.847,Z 849.946,A -85,B 0,C 180,E1 -3220.663,E2 -3220.663} C_VEL
LIN {X 0,Y 551.738,Z 855.422,A -85,B 0,C 180,E1 -3221.815,E2 -3221.815} C_VEL
LIN {X 0,Y 551.745,Z 859.634,A -85,B 0,C 180,E1 -3222.964,E2 -3222.964} C_VEL
LIN {X 0,Y 551.678,Z 861.846,A -85,B 0,C 180,E1 -3223.724,E2 -3223.724} C_VEL
LIN {X 0,Y 551.622,Z 863.517,A -85,B 0,C 180,E1 -3224.481,E2 -3224.481} C_VEL
LIN {X 0,Y 551.674,Z 865.575,A -85,B 0,C 180,E1 -3225.992,E2 -3225.992} C_VEL
LIN {X 0,Y 551.659,Z 865.93,A -85,B 0,C 180,E1 -3226.743,E2 -3226.743} C_VEL
LIN {X 0,Y 551.675,Z 865.468,A -85,B 0,C 180,E1 -3228.239,E2 -3228.239} C_VEL
LIN {X 0,Y 551.705,Z 864.556,A -85,B 0,C 180,E1 -3228.984,E2 -3228.984} C_VEL
LIN {X 0,Y 551.688,Z 861.6,A -85,B 0,C 180,E1 -3230.467,E2 -3230.467} C_VEL
LIN {X 0,Y 551.738,Z 858.184,A -85,B 0,C 180,E1 -3231.576,E2 -3231.576} C_VEL
LIN {X 0,Y 551.801,Z 853.688,A -85,B 0,C 180,E1 -3232.683,E2 -3232.683} C_VEL
LIN {X 0,Y 551.858,Z 847.271,A -85,B 0,C 180,E1 -3233.901,E2 -3233.901} C_VEL
LIN {X 0,Y 551.893,Z 840.853,A -85,B 0,C 180,E1 -3234.886,E2 -3234.886} C_VEL
LIN {X 0,Y 552.052,Z 833.623,A -85,B 0,C 180,E1 -3235.802,E2 -3235.802} C_VEL
LIN {X 0,Y 552.195,Z 824.924,A -85,B 0,C 180,E1 -3236.717,E2 -3236.717} C_VEL
LIN {X 0,Y 552.344,Z 816.574,A -85,B 0,C 180,E1 -3237.447,E2 -3237.447} C_VEL
LIN {X 0,Y 552.497,Z 807.868,A -85,B 0,C 180,E1 -3238.086,E2 -3238.086} C_VEL
LIN {X 0,Y 552.619,Z 798.932,A -85,B 0,C 180,E1 -3238.633,E2 -3238.633} C_VEL
LIN {X 0,Y 552.827,Z 788.77,A -85,B 0,C 180,E1 -3239.135,E2 -3239.135} C_VEL
LIN {X 0,Y 552.984,Z 778.06,A -85,B 0,C 180,E1 -3239.545,E2 -3239.545} C_VEL
LIN {X 0,Y 553.044,Z 766.536,A -85,B 0,C 180,E1 -3239.863,E2 -3239.863} C_VEL
LIN {X 0,Y 553.187,Z 753.295,A -85,B 0,C 180,E1 -3240.091,E2 -3240.091} C_VEL
LIN {X 0,Y 553.341,Z 687.781,A -85,B 0,C 180,E1 -3240.944,E2 -3240.944} C_VEL
LIN {X 0,Y 552.322,Z 684.407,A -85,B 0,C 180,E1 -3241.048,E2 -3241.048} C_VEL
LIN {X 0,Y 552.19,Z 683.75,A -85,B 0,C 180,E1 -3241.185,E2 -3241.185} C_VEL
LIN {X 0,Y 552.206,Z 683.698,A -85,B 0,C 180,E1 -3242.918,E2 -3242.918} C_VEL
LIN {X 0,Y 552.195,Z 683.704,A -85,B 0,C 180,E1 -3245.844,E2 -3245.844} C_VEL
LIN {X 0,Y 552.146,Z 683.704,A -85,B 0,C 180,E1 -3248.786,E2 -3248.786} C_VEL
LIN {X 0,Y 552.168,Z 683.702,A -85,B 0,C 180,E1 -3251.75,E2 -3251.75} C_VEL
LIN {X 0,Y 552.143,Z 683.706,A -85,B 0,C 180,E1 -3254.748,E2 -3254.748} C_VEL
LIN {X 0,Y 552.102,Z 683.709,A -85,B 0,C 180,E1 -3257.789,E2 -3257.789} C_VEL
LIN {X 0,Y 552.133,Z 683.707,A -85,B 0,C 180,E1 -3260.101,E2 -3260.101} C_VEL
LIN {X 0,Y 552.097,Z 683.716,A -85,B 0,C 180,E1 -3262.451,E2 -3262.451} C_VEL
LIN {X 0,Y 552.144,Z 683.703,A -85,B 0,C 180,E1 -3265.346,E2 -3265.346} C_VEL
LIN {X 0,Y 552.084,Z 683.711,A -85,B 0,C 180,E1 -3268.1,E2 -3268.1} C_VEL
LIN {X 0,Y 552.108,Z 683.713,A -85,B 0,C 180,E1 -3270.609,E2 -3270.609} C_VEL
LIN {X 0,Y 552.112,Z 683.712,A -85,B 0,C 180,E1 -3273.186,E2 -3273.186} C_VEL
LIN {X 0,Y 552.091,Z 683.709,A -85,B 0,C 180,E1 -3275.843,E2 -3275.843} C_VEL
LIN {X 0,Y 552.122,Z 683.707,A -85,B 0,C 180,E1 -3278.589,E2 -3278.589} C_VEL
LIN {X 0,Y 552.126,Z 683.71,A -85,B 0,C 180,E1 -3281.446,E2 -3281.446} C_VEL
LIN {X 0,Y 552.095,Z 683.709,A -85,B 0,C 180,E1 -3284.531,E2 -3284.531} C_VEL
LIN {X 0,Y 552.136,Z 683.71,A -85,B 0,C 180,E1 -3287.584,E2 -3287.584} C_VEL
LIN {X 0,Y 552.133,Z 683.703,A -85,B 0,C 180,E1 -3290.472,E2 -3290.472} C_VEL
LIN {X 0,Y 552.105,Z 683.712,A -85,B 0,C 180,E1 -3293.318,E2 -3293.318} C_VEL
LIN {X 0,Y 552.107,Z 683.714,A -85,B 0,C 180,E1 -3295.937,E2 -3295.937} C_VEL
LIN {X 0,Y 552.126,Z 683.707,A -85,B 0,C 180,E1 -3298.54,E2 -3298.54} C_VEL
LIN {X 0,Y 552.103,Z 683.712,A -85,B 0,C 180,E1 -3301.443,E2 -3301.443} C_VEL
LIN {X 0,Y 552.143,Z 683.933,A -85,B 0,C 180,E1 -3302.002,E2 -3302.002} C_VEL
LIN {X 0,Y 554.507,Z 693.884,A -85,B 0,C 180,E1 -3303.259,E2 -3303.259} C_VEL
LIN {X 0,Y 554.234,Z 713.228,A -85,B 0,C 180,E1 -3305.482,E2 -3305.482} C_VEL
LIN {X 0,Y 553.652,Z 739.956,A -85,B 0,C 180,E1 -3308.595,E2 -3308.595} C_VEL
LIN {X 0,Y 553.148,Z 766.852,A -85,B 0,C 180,E1 -3311.671,E2 -3311.671} C_VEL
LIN {X 0,Y 552.689,Z 795.765,A -85,B 0,C 180,E1 -3314.926,E2 -3314.926} C_VEL
LIN {X 0,Y 552.615,Z 801.878,A -85,B 0,C 180,E1 -3315.593,E2 -3315.593} C_VEL
LIN {X 0,Y 553.438,Z 809.431,A -85,B 0,C 180,E1 -3315.732,E2 -3315.732} C_VEL
LIN {X 0,Y 553.122,Z 911.896,A -85,B 0,C 180,E1 -3317.082,E2 -3317.082} C_VEL
LIN {X 0,Y 553.029,Z 924.423,A -85,B 0,C 180,E1 -3317.383,E2 -3317.383} C_VEL
LIN {X 0,Y 552.851,Z 937.343,A -85,B 0,C 180,E1 -3317.845,E2 -3317.845} C_VEL
LIN {X 0,Y 552.691,Z 949.654,A -85,B 0,C 180,E1 -3318.448,E2 -3318.448} C_VEL
LIN {X 0,Y 552.502,Z 961.186,A -85,B 0,C 180,E1 -3319.185,E2 -3319.185} C_VEL
LIN {X 0,Y 552.296,Z 971.59,A -85,B 0,C 180,E1 -3320.015,E2 -3320.015} C_VEL
LIN {X 0,Y 552.126,Z 980.064,A -85,B 0,C 180,E1 -3320.844,E2 -3320.844} C_VEL
LIN {X 0,Y 552.009,Z 987.952,A -85,B 0,C 180,E1 -3321.764,E2 -3321.764} C_VEL
LIN {X 0,Y 551.891,Z 995.614,A -85,B 0,C 180,E1 -3322.867,E2 -3322.867} C_VEL
LIN {X 0,Y 551.869,Z 1002.675,A -85,B 0,C 180,E1 -3324.152,E2 -3324.152} C_VEL
LIN {X 0,Y 551.725,Z 1007.368,A -85,B 0,C 180,E1 -3325.25,E2 -3325.25} C_VEL
LIN {X 0,Y 551.75,Z 1010.954,A -85,B 0,C 180,E1 -3326.347,E2 -3326.347} C_VEL
LIN {X 0,Y 551.724,Z 1012.806,A -85,B 0,C 180,E1 -3327.078,E2 -3327.078} C_VEL
LIN {X 0,Y 551.645,Z 1015.184,A -85,B 0,C 180,E1 -3328.539,E2 -3328.539} C_VEL
LIN {X 0,Y 551.64,Z 1016,A -85,B 0,C 180,E1 -3329.999,E2 -3329.999} C_VEL
LIN {X 0,Y 551.644,Z 1015.187,A -85,B 0,C 180,E1 -3331.459,E2 -3331.459} C_VEL
LIN {X 0,Y 551.723,Z 1012.812,A -85,B 0,C 180,E1 -3332.92,E2 -3332.92} C_VEL
LIN {X 0,Y 551.763,Z 1009.899,A -85,B 0,C 180,E1 -3334.016,E2 -3334.016} C_VEL
LIN {X 0,Y 551.723,Z 1005.953,A -85,B 0,C 180,E1 -3335.115,E2 -3335.115} C_VEL
LIN {X 0,Y 551.816,Z 1000.122,A -85,B 0,C 180,E1 -3336.354,E2 -3336.354} C_VEL
LIN {X 0,Y 551.925,Z 993.245,A -85,B 0,C 180,E1 -3337.498,E2 -3337.498} C_VEL
LIN {X 0,Y 552.072,Z 985,A -85,B 0,C 180,E1 -3338.601,E2 -3338.601} C_VEL
LIN {X 0,Y 552.241,Z 974.613,A -85,B 0,C 180,E1 -3339.707,E2 -3339.707} C_VEL
LIN {X 0,Y 552.429,Z 963.762,A -85,B 0,C 180,E1 -3340.629,E2 -3340.629} C_VEL
LIN {X 0,Y 552.628,Z 952.92,A -85,B 0,C 180,E1 -3341.361,E2 -3341.361} C_VEL
LIN {X 0,Y 552.816,Z 940.53,A -85,B 0,C 180,E1 -3342.014,E2 -3342.014} C_VEL
LIN {X 0,Y 552.949,Z 928.903,A -85,B 0,C 180,E1 -3342.477,E2 -3342.477} C_VEL
LIN {X 0,Y 553.077,Z 916.563,A -85,B 0,C 180,E1 -3342.824,E2 -3342.824} C_VEL
LIN {X 0,Y 553.167,Z 900.825,A -85,B 0,C 180,E1 -3343.079,E2 -3343.079} C_VEL
LIN {X 0,Y 553.298,Z 807.143,A -85,B 0,C 180,E1 -3344.301,E2 -3344.301} C_VEL
LIN {X 0,Y 552.6,Z 801.916,A -85,B 0,C 180,E1 -3344.405,E2 -3344.405} C_VEL
LIN {X 0,Y 553.007,Z 774.403,A -85,B 0,C 180,E1 -3347.475,E2 -3347.475} C_VEL
LIN {X 0,Y 553.526,Z 746.7,A -85,B 0,C 180,E1 -3350.629,E2 -3350.629} C_VEL
LIN {X 0,Y 554.12,Z 719.804,A -85,B 0,C 180,E1 -3353.745,E2 -3353.745} C_VEL
LIN {X 0,Y 554.492,Z 698.732,A -85,B 0,C 180,E1 -3356.178,E2 -3356.178} C_VEL
LIN {X 0,Y 554.498,Z 693.794,A -85,B 0,C 180,E1 -3356.739,E2 -3356.739} C_VEL
LIN {X 0,Y 552.184,Z 683.894,A -85,B 0,C 180,E1 -3357.989,E2 -3357.989} C_VEL
LIN {X 0,Y 552.099,Z 683.714,A -85,B 0,C 180,E1 -3360.608,E2 -3360.608} C_VEL
LIN {X 0,Y 552.107,Z 683.708,A -85,B 0,C 180,E1 -3363.185,E2 -3363.185} C_VEL
LIN {X 0,Y 552.08,Z 683.713,A -85,B 0,C 180,E1 -3365.842,E2 -3365.842} C_VEL
LIN {X 0,Y 552.111,Z 683.715,A -85,B 0,C 180,E1 -3368.588,E2 -3368.588} C_VEL
LIN {X 0,Y 552.114,Z 683.706,A -85,B 0,C 180,E1 -3371.445,E2 -3371.445} C_VEL
LIN {X 0,Y 552.088,Z 683.715,A -85,B 0,C 180,E1 -3374.531,E2 -3374.531} C_VEL
LIN {X 0,Y 552.123,Z 683.705,A -85,B 0,C 180,E1 -3377.583,E2 -3377.583} C_VEL
LIN {X 0,Y 552.126,Z 683.704,A -85,B 0,C 180,E1 -3380.472,E2 -3380.472} C_VEL
LIN {X 0,Y 552.106,Z 683.71,A -85,B 0,C 180,E1 -3383.315,E2 -3383.315} C_VEL
LIN {X 0,Y 552.122,Z 683.704,A -85,B 0,C 180,E1 -3385.939,E2 -3385.939} C_VEL
LIN {X 0,Y 552.108,Z 683.707,A -85,B 0,C 180,E1 -3388.54,E2 -3388.54} C_VEL
LIN {X 0,Y 552.117,Z 683.713,A -85,B 0,C 180,E1 -3391.437,E2 -3391.437} C_VEL
LIN {X 0,Y 552.126,Z 683.703,A -85,B 0,C 180,E1 -3394.356,E2 -3394.356} C_VEL
LIN {X 0,Y 552.099,Z 683.707,A -85,B 0,C 180,E1 -3396.758,E2 -3396.758} C_VEL
LIN {X 0,Y 552.11,Z 683.707,A -85,B 0,C 180,E1 -3399.119,E2 -3399.119} C_VEL
LIN {X 0,Y 552.117,Z 683.711,A -85,B 0,C 180,E1 -3401.444,E2 -3401.444} C_VEL
LIN {X 0,Y 552.104,Z 683.715,A -85,B 0,C 180,E1 -3403.737,E2 -3403.737} C_VEL
LIN {X 0,Y 552.124,Z 683.71,A -85,B 0,C 180,E1 -3406.004,E2 -3406.004} C_VEL
LIN {X 0,Y 552.15,Z 683.701,A -85,B 0,C 180,E1 -3408.993,E2 -3408.993} C_VEL
LIN {X 0,Y 552.15,Z 683.707,A -85,B 0,C 180,E1 -3411.951,E2 -3411.951} C_VEL
LIN {X 0,Y 552.218,Z 683.692,A -85,B 0,C 180,E1 -3414.889,E2 -3414.889} C_VEL
LIN {X 0,Y 552.207,Z 683.696,A -85,B 0,C 180,E1 -3417.812,E2 -3417.812} C_VEL
LIN {X 0,Y 552.236,Z 683.694,A -85,B 0,C 180,E1 -3420.729,E2 -3420.729} C_VEL
LIN {X 0,Y 552.2,Z 683.697,A -85,B 0,C 180,E1 -3422.918,E2 -3422.918} C_VEL
LIN {X 0,Y 552.185,Z 683.697,A -85,B 0,C 180,E1 -3425.844,E2 -3425.844} C_VEL
LIN {X 0,Y 552.152,Z 683.709,A -85,B 0,C 180,E1 -3428.786,E2 -3428.786} C_VEL
LIN {X 0,Y 552.153,Z 683.7,A -85,B 0,C 180,E1 -3431.751,E2 -3431.751} C_VEL
LIN {X 0,Y 552.125,Z 683.712,A -85,B 0,C 180,E1 -3434.749,E2 -3434.749} C_VEL
LIN {X 0,Y 552.087,Z 683.709,A -85,B 0,C 180,E1 -3437.789,E2 -3437.789} C_VEL
LIN {X 0,Y 552.118,Z 683.704,A -85,B 0,C 180,E1 -3440.102,E2 -3440.102} C_VEL
LIN {X 0,Y 552.081,Z 683.709,A -85,B 0,C 180,E1 -3442.452,E2 -3442.452} C_VEL
LIN {X 0,Y 552.106,Z 683.711,A -85,B 0,C 180,E1 -3445.646,E2 -3445.646} C_VEL
LIN {X 0,Y 552.086,Z 683.707,A -85,B 0,C 180,E1 -3448.1,E2 -3448.1} C_VEL
LIN {X 0,Y 552.091,Z 683.709,A -85,B 0,C 180,E1 -3450.627,E2 -3450.627} C_VEL
LIN {X 0,Y 552.114,Z 683.708,A -85,B 0,C 180,E1 -3453.186,E2 -3453.186} C_VEL
LIN {X 0,Y 552.104,Z 683.708,A -85,B 0,C 180,E1 -3453.806,E2 -3453.806} C_VEL
LIN {X 0,Y 551.468,Z 683.791,A -85,B 0,C 180,E1 -3454.415,E2 -3454.415} C_VEL
LIN {X 0,Y 548.645,Z 684.145,A -85,B 0,C 180,E1 -3455.403,E2 -3455.403} C_VEL
LIN {X 0,Y 546.224,Z 684.441,A -85,B 0,C 180,E1 -3456.198,E2 -3456.198} C_VEL
LIN {X 0,Y 545.155,Z 684.573,A -85,B 0,C 180,E1 -3456.812,E2 -3456.812} C_VEL
LIN {X 0,Y 545.054,Z 684.586,A -85,B 0,C 180,E1 -3457.02,E2 -3457.02} C_VEL
LIN {X 0,Y 545.058,Z 684.589,A -85,B 0,C 180,E1 -3460.144,E2 -3460.144} C_VEL
LIN {X 0,Y 545.072,Z 684.583,A -85,B 0,C 180,E1 -3463.108,E2 -3463.108} C_VEL
LIN {X 0,Y 545.043,Z 684.591,A -85,B 0,C 180,E1 -3466.228,E2 -3466.228} C_VEL
LIN {X 0,Y 545.075,Z 684.585,A -85,B 0,C 180,E1 -3468.887,E2 -3468.887} C_VEL
LIN {X 0,Y 545.124,Z 684.789,A -85,B 0,C 180,E1 -3470.765,E2 -3470.765} C_VEL
LIN {X 0,Y 545.386,Z 685.988,A -85,B 0,C 180,E1 -3470.885,E2 -3470.885} C_VEL
LIN {X 0,Y 546.44,Z 689.135,A -85,B 0,C 180,E1 -3470.961,E2 -3470.961} C_VEL
LIN {X 0,Y 546.243,Z 764.36,A -85,B 0,C 180,E1 -3471.98,E2 -3471.98} C_VEL
LIN {X 0,Y 546.138,Z 777.756,A -85,B 0,C 180,E1 -3472.321,E2 -3472.321} C_VEL
LIN {X 0,Y 545.979,Z 789.745,A -85,B 0,C 180,E1 -3472.773,E2 -3472.773} C_VEL
LIN {X 0,Y 545.807,Z 800.865,A -85,B 0,C 180,E1 -3473.336,E2 -3473.336} C_VEL
LIN {X 0,Y 545.611,Z 812.422,A -85,B 0,C 180,E1 -3474.092,E2 -3474.092} C_VEL
LIN {X 0,Y 545.38,Z 822.294,A -85,B 0,C 180,E1 -3474.898,E2 -3474.898} C_VEL
LIN {X 0,Y 545.169,Z 832.113,A -85,B 0,C 180,E1 -3475.892,E2 -3475.892} C_VEL
LIN {X 0,Y 544.948,Z 840.583,A -85,B 0,C 180,E1 -3476.96,E2 -3476.96} C_VEL
LIN {X 0,Y 544.849,Z 847.706,A -85,B 0,C 180,E1 -3478.073,E2 -3478.073} C_VEL
LIN {X 0,Y 544.737,Z 854.206,A -85,B 0,C 180,E1 -3479.363,E2 -3479.363} C_VEL
LIN {X 0,Y 544.682,Z 859.059,A -85,B 0,C 180,E1 -3480.64,E2 -3480.64} C_VEL
LIN {X 0,Y 544.617,Z 861.544,A -85,B 0,C 180,E1 -3481.481,E2 -3481.481} C_VEL
LIN {X 0,Y 544.553,Z 864.479,A -85,B 0,C 180,E1 -3482.939,E2 -3482.939} C_VEL
LIN {X 0,Y 544.555,Z 865.65,A -85,B 0,C 180,E1 -3483.974,E2 -3483.974} C_VEL
LIN {X 0,Y 544.552,Z 866.014,A -85,B 0,C 180,E1 -3484.794,E2 -3484.794} C_VEL
LIN {X 0,Y 544.539,Z 865.949,A -85,B 0,C 180,E1 -3485.608,E2 -3485.608} C_VEL
LIN {X 0,Y 544.557,Z 865.375,A -85,B 0,C 180,E1 -3486.418,E2 -3486.418} C_VEL
LIN {X 0,Y 544.551,Z 864.366,A -85,B 0,C 180,E1 -3487.222,E2 -3487.222} C_VEL
LIN {X 0,Y 544.59,Z 862.256,A -85,B 0,C 180,E1 -3488.307,E2 -3488.307} C_VEL
LIN {X 0,Y 544.673,Z 858.518,A -85,B 0,C 180,E1 -3489.613,E2 -3489.613} C_VEL
LIN {X 0,Y 544.776,Z 853.891,A -85,B 0,C 180,E1 -3490.795,E2 -3490.795} C_VEL
LIN {X 0,Y 544.851,Z 847.966,A -85,B 0,C 180,E1 -3491.968,E2 -3491.968} C_VEL
LIN {X 0,Y 544.946,Z 840.526,A -85,B 0,C 180,E1 -3493.133,E2 -3493.133} C_VEL
LIN {X 0,Y 545.15,Z 832.889,A -85,B 0,C 180,E1 -3494.102,E2 -3494.102} C_VEL
LIN {X 0,Y 545.328,Z 823.648,A -85,B 0,C 180,E1 -3495.064,E2 -3495.064} C_VEL
LIN {X 0,Y 545.534,Z 813.324,A -85,B 0,C 180,E1 -3495.928,E2 -3495.928} C_VEL
LIN {X 0,Y 545.778,Z 801.786,A -85,B 0,C 180,E1 -3496.694,E2 -3496.694} C_VEL
LIN {X 0,Y 545.991,Z 789.711,A -85,B 0,C 180,E1 -3497.314,E2 -3497.314} C_VEL
LIN {X 0,Y 546.132,Z 777.14,A -85,B 0,C 180,E1 -3497.785,E2 -3497.785} C_VEL
LIN {X 0,Y 546.281,Z 763.615,A -85,B 0,C 180,E1 -3498.122,E2 -3498.122} C_VEL
LIN {X 0,Y 546.354,Z 688.785,A -85,B 0,C 180,E1 -3499.134,E2 -3499.134} C_VEL
LIN {X 0,Y 545.265,Z 685.496,A -85,B 0,C 180,E1 -3499.23,E2 -3499.23} C_VEL
LIN {X 0,Y 545.102,Z 684.65,A -85,B 0,C 180,E1 -3499.367,E2 -3499.367} C_VEL
LIN {X 0,Y 545.07,Z 684.59,A -85,B 0,C 180,E1 -3501.847,E2 -3501.847} C_VEL
LIN {X 0,Y 545.164,Z 684.573,A -85,B 0,C 180,E1 -3504.824,E2 -3504.824} C_VEL
LIN {X 0,Y 545.192,Z 684.573,A -85,B 0,C 180,E1 -3507.785,E2 -3507.785} C_VEL
LIN {X 0,Y 545.194,Z 684.575,A -85,B 0,C 180,E1 -3510.001,E2 -3510.001} C_VEL
LIN {X 0,Y 545.146,Z 684.576,A -85,B 0,C 180,E1 -3512.957,E2 -3512.957} C_VEL
LIN {X 0,Y 545.125,Z 684.579,A -85,B 0,C 180,E1 -3515.921,E2 -3515.921} C_VEL
LIN {X 0,Y 545.07,Z 684.587,A -85,B 0,C 180,E1 -3518.902,E2 -3518.902} C_VEL
LIN {X 0,Y 545.058,Z 684.585,A -85,B 0,C 180,E1 -3521.907,E2 -3521.907} C_VEL
LIN {X 0,Y 545.083,Z 684.586,A -85,B 0,C 180,E1 -3524.945,E2 -3524.945} C_VEL
LIN {X 0,Y 545.051,Z 684.586,A -85,B 0,C 180,E1 -3528.028,E2 -3528.028} C_VEL
LIN {X 0,Y 545.052,Z 684.584,A -85,B 0,C 180,E1 -3530.375,E2 -3530.375} C_VEL
LIN {X 0,Y 545.03,Z 684.594,A -85,B 0,C 180,E1 -3532.759,E2 -3532.759} C_VEL
LIN {X 0,Y 545.011,Z 684.589,A -85,B 0,C 180,E1 -3535.489,E2 -3535.489} C_VEL
LIN {X 0,Y 545.002,Z 684.591,A -85,B 0,C 180,E1 -3537.662,E2 -3537.662} C_VEL
LIN {X 0,Y 545.026,Z 684.588,A -85,B 0,C 180,E1 -3540.236,E2 -3540.236} C_VEL
LIN {X 0,Y 545.057,Z 684.59,A -85,B 0,C 180,E1 -3543.058,E2 -3543.058} C_VEL
LIN {X 0,Y 545.017,Z 684.59,A -85,B 0,C 180,E1 -3545.67,E2 -3545.67} C_VEL
LIN {X 0,Y 545.02,Z 684.589,A -85,B 0,C 180,E1 -3548.241,E2 -3548.241} C_VEL
LIN {X 0,Y 544.999,Z 684.595,A -85,B 0,C 180,E1 -3551.123,E2 -3551.123} C_VEL
LIN {X 0,Y 545.029,Z 684.59,A -85,B 0,C 180,E1 -3554.133,E2 -3554.133} C_VEL
LIN {X 0,Y 545.004,Z 684.591,A -85,B 0,C 180,E1 -3556.886,E2 -3556.886} C_VEL
LIN {X 0,Y 545.01,Z 684.6,A -85,B 0,C 180,E1 -3559.852,E2 -3559.852} C_VEL
LIN {X 0,Y 544.98,Z 684.595,A -85,B 0,C 180,E1 -3562.691,E2 -3562.691} C_VEL
LIN {X 0,Y 545.051,Z 684.59,A -85,B 0,C 180,E1 -3565.613,E2 -3565.613} C_VEL
LIN {X 0,Y 545.049,Z 684.593,A -85,B 0,C 180,E1 -3568.324,E2 -3568.324} C_VEL
LIN {X 0,Y 545.034,Z 684.593,A -85,B 0,C 180,E1 -3571.503,E2 -3571.503} C_VEL
LIN {X 0,Y 545.064,Z 684.741,A -85,B 0,C 180,E1 -3572.77,E2 -3572.77} C_VEL
LIN {X 0,Y 545.309,Z 685.813,A -85,B 0,C 180,E1 -3572.902,E2 -3572.902} C_VEL
LIN {X 0,Y 546.378,Z 689.132,A -85,B 0,C 180,E1 -3572.984,E2 -3572.984} C_VEL
LIN {X 0,Y 546.209,Z 761.429,A -85,B 0,C 180,E1 -3573.954,E2 -3573.954} C_VEL
LIN {X 0,Y 546.068,Z 773.503,A -85,B 0,C 180,E1 -3574.241,E2 -3574.241} C_VEL
LIN {X 0,Y 545.925,Z 784.505,A -85,B 0,C 180,E1 -3574.62,E2 -3574.62} C_VEL
LIN {X 0,Y 545.769,Z 794.193,A -85,B 0,C 180,E1 -3575.056,E2 -3575.056} C_VEL
LIN {X 0,Y 545.572,Z 804.723,A -85,B 0,C 180,E1 -3575.655,E2 -3575.655} C_VEL
LIN {X 0,Y 545.433,Z 813.607,A -85,B 0,C 180,E1 -3576.274,E2 -3576.274} C_VEL
LIN {X 0,Y 545.198,Z 822.818,A -85,B 0,C 180,E1 -3577.049,E2 -3577.049} C_VEL
LIN {X 0,Y 545.059,Z 830.686,A -85,B 0,C 180,E1 -3577.842,E2 -3577.842} C_VEL
LIN {X 0,Y 544.962,Z 837.525,A -85,B 0,C 180,E1 -3578.655,E2 -3578.655} C_VEL
LIN {X 0,Y 544.799,Z 844.301,A -85,B 0,C 180,E1 -3579.616,E2 -3579.616} C_VEL
LIN {X 0,Y 544.788,Z 849.018,A -85,B 0,C 180,E1 -3580.402,E2 -3580.402} C_VEL
LIN {X 0,Y 544.666,Z 854.71,A -85,B 0,C 180,E1 -3581.571,E2 -3581.571} C_VEL
LIN {X 0,Y 544.658,Z 859.092,A -85,B 0,C 180,E1 -3582.735,E2 -3582.735} C_VEL
LIN {X 0,Y 544.613,Z 861.411,A -85,B 0,C 180,E1 -3583.507,E2 -3583.507} C_VEL
LIN {X 0,Y 544.517,Z 864.493,A -85,B 0,C 180,E1 -3585.04,E2 -3585.04} C_VEL
LIN {X 0,Y 544.59,Z 865.435,A -85,B 0,C 180,E1 -3585.806,E2 -3585.806} C_VEL
LIN {X 0,Y 544.57,Z 865.933,A -85,B 0,C 180,E1 -3587.326,E2 -3587.326} C_VEL
LIN {X 0,Y 544.569,Z 865.596,A -85,B 0,C 180,E1 -3588.083,E2 -3588.083} C_VEL
LIN {X 0,Y 544.583,Z 863.62,A -85,B 0,C 180,E1 -3589.591,E2 -3589.591} C_VEL
LIN {X 0,Y 544.61,Z 861.028,A -85,B 0,C 180,E1 -3590.717,E2 -3590.717} C_VEL
LIN {X 0,Y 544.658,Z 857.42,A -85,B 0,C 180,E1 -3591.84,E2 -3591.84} C_VEL
LIN {X 0,Y 544.734,Z 852.7,A -85,B 0,C 180,E1 -3592.96,E2 -3592.96} C_VEL
LIN {X 0,Y 544.827,Z 846.736,A -85,B 0,C 180,E1 -3594.077,E2 -3594.077} C_VEL
LIN {X 0,Y 544.863,Z 840.715,A -85,B 0,C 180,E1 -3595.005,E2 -3595.005} C_VEL
LIN {X 0,Y 544.989,Z 833.473,A -85,B 0,C 180,E1 -3595.933,E2 -3595.933} C_VEL
LIN {X 0,Y 545.12,Z 826.689,A -85,B 0,C 180,E1 -3596.674,E2 -3596.674} C_VEL
LIN {X 0,Y 545.334,Z 817.512,A -85,B 0,C 180,E1 -3597.507,E2 -3597.507} C_VEL
LIN {X 0,Y 545.5,Z 807.603,A -85,B 0,C 180,E1 -3598.246,E2 -3598.246} C_VEL
LIN {X 0,Y 545.656,Z 798.598,A -85,B 0,C 180,E1 -3598.801,E2 -3598.801} C_VEL
LIN {X 0,Y 545.887,Z 788.342,A -85,B 0,C 180,E1 -3599.308,E2 -3599.308} C_VEL
LIN {X 0,Y 546.039,Z 777.5,A -85,B 0,C 180,E1 -3599.723,E2 -3599.723} C_VEL
LIN {X 0,Y 546.142,Z 766.741,A -85,B 0,C 180,E1 -3600.023,E2 -3600.023} C_VEL
LIN {X 0,Y 546.262,Z 755.487,A -85,B 0,C 180,E1 -3600.23,E2 -3600.23} C_VEL
LIN {X 0,Y 546.37,Z 688.793,A -85,B 0,C 180,E1 -3601.111,E2 -3601.111} C_VEL
LIN {X 0,Y 545.328,Z 685.554,A -85,B 0,C 180,E1 -3601.2,E2 -3601.2} C_VEL
LIN {X 0,Y 545.112,Z 684.656,A -85,B 0,C 180,E1 -3601.339,E2 -3601.339} C_VEL
LIN {X 0,Y 545.173,Z 684.575,A -85,B 0,C 180,E1 -3602.956,E2 -3602.956} C_VEL
LIN {X 0,Y 545.165,Z 684.58,A -85,B 0,C 180,E1 -3605.919,E2 -3605.919} C_VEL
LIN {X 0,Y 545.107,Z 684.58,A -85,B 0,C 180,E1 -3608.9,E2 -3608.9} C_VEL
LIN {X 0,Y 545.111,Z 684.583,A -85,B 0,C 180,E1 -3611.905,E2 -3611.905} C_VEL
LIN {X 0,Y 545.092,Z 684.583,A -85,B 0,C 180,E1 -3614.943,E2 -3614.943} C_VEL
LIN {X 0,Y 545.074,Z 684.586,A -85,B 0,C 180,E1 -3618.026,E2 -3618.026} C_VEL
LIN {X 0,Y 545.099,Z 684.588,A -85,B 0,C 180,E1 -3620.372,E2 -3620.372} C_VEL
LIN {X 0,Y 545.084,Z 684.581,A -85,B 0,C 180,E1 -3623.559,E2 -3623.559} C_VEL
LIN {X 0,Y 545.081,Z 684.583,A -85,B 0,C 180,E1 -3626.001,E2 -3626.001} C_VEL
LIN {X 0,Y 545.076,Z 684.591,A -85,B 0,C 180,E1 -3628.744,E2 -3628.744} C_VEL
LIN {X 0,Y 545.064,Z 684.584,A -85,B 0,C 180,E1 -3631.678,E2 -3631.678} C_VEL
LIN {X 0,Y 545.065,Z 684.587,A -85,B 0,C 180,E1 -3634.564,E2 -3634.564} C_VEL
LIN {X 0,Y 545.042,Z 684.593,A -85,B 0,C 180,E1 -3637.304,E2 -3637.304} C_VEL
LIN {X 0,Y 545.071,Z 684.583,A -85,B 0,C 180,E1 -3640.142,E2 -3640.142} C_VEL
LIN {X 0,Y 545.085,Z 684.589,A -85,B 0,C 180,E1 -3643.106,E2 -3643.106} C_VEL
LIN {X 0,Y 545.055,Z 684.585,A -85,B 0,C 180,E1 -3646.226,E2 -3646.226} C_VEL
LIN {X 0,Y 545.087,Z 684.583,A -85,B 0,C 180,E1 -3648.885,E2 -3648.885} C_VEL
LIN {X 0,Y 545.052,Z 684.59,A -85,B 0,C 180,E1 -3651.864,E2 -3651.864} C_VEL
LIN {X 0,Y 545.035,Z 684.588,A -85,B 0,C 180,E1 -3654.53,E2 -3654.53} C_VEL
LIN {X 0,Y 545.07,Z 684.587,A -85,B 0,C 180,E1 -3657.211,E2 -3657.211} C_VEL
LIN {X 0,Y 545.068,Z 684.593,A -85,B 0,C 180,E1 -3659.81,E2 -3659.81} C_VEL
LIN {X 0,Y 545.098,Z 684.817,A -85,B 0,C 180,E1 -3661.808,E2 -3661.808} C_VEL
LIN {X 0,Y 547.551,Z 695.004,A -85,B 0,C 180,E1 -3663.115,E2 -3663.115} C_VEL
LIN {X 0,Y 547.548,Z 705.478,A -85,B 0,C 180,E1 -3664.329,E2 -3664.329} C_VEL
LIN {X 0,Y 547.024,Z 729.87,A -85,B 0,C 180,E1 -3667.129,E2 -3667.129} C_VEL
LIN {X 0,Y 546.554,Z 751.723,A -85,B 0,C 180,E1 -3669.684,E2 -3669.684} C_VEL
LIN {X 0,Y 546.066,Z 776.887,A -85,B 0,C 180,E1 -3672.582,E2 -3672.582} C_VEL
LIN {X 0,Y 545.629,Z 801.976,A -85,B 0,C 180,E1 -3675.41,E2 -3675.41} C_VEL
LIN {X 0,Y 546.568,Z 809.726,A -85,B 0,C 180,E1 -3675.553,E2 -3675.553} C_VEL
LIN {X 0,Y 546.214,Z 911.896,A -85,B 0,C 180,E1 -3676.915,E2 -3676.915} C_VEL
LIN {X 0,Y 546.097,Z 924.423,A -85,B 0,C 180,E1 -3677.22,E2 -3677.22} C_VEL
LIN {X 0,Y 545.9,Z 937.344,A -85,B 0,C 180,E1 -3677.687,E2 -3677.687} C_VEL
LIN {X 0,Y 545.733,Z 949.653,A -85,B 0,C 180,E1 -3678.299,E2 -3678.299} C_VEL
LIN {X 0,Y 545.525,Z 961.184,A -85,B 0,C 180,E1 -3679.045,E2 -3679.045} C_VEL
LIN {X 0,Y 545.258,Z 971.591,A -85,B 0,C 180,E1 -3679.884,E2 -3679.884} C_VEL
LIN {X 0,Y 545.085,Z 980.073,A -85,B 0,C 180,E1 -3680.724,E2 -3680.724} C_VEL
LIN {X 0,Y 544.972,Z 987.952,A -85,B 0,C 180,E1 -3681.657,E2 -3681.657} C_VEL
LIN {X 0,Y 544.825,Z 995.615,A -85,B 0,C 180,E1 -3682.774,E2 -3682.774} C_VEL
LIN {X 0,Y 544.779,Z 1002.675,A -85,B 0,C 180,E1 -3684.075,E2 -3684.075} C_VEL
LIN {X 0,Y 544.629,Z 1007.368,A -85,B 0,C 180,E1 -3685.187,E2 -3685.187} C_VEL
LIN {X 0,Y 544.669,Z 1010.955,A -85,B 0,C 180,E1 -3686.3,E2 -3686.3} C_VEL
LIN {X 0,Y 544.65,Z 1012.805,A -85,B 0,C 180,E1 -3687.04,E2 -3687.04} C_VEL
LIN {X 0,Y 544.545,Z 1015.183,A -85,B 0,C 180,E1 -3688.52,E2 -3688.52} C_VEL
LIN {X 0,Y 544.541,Z 1016,A -85,B 0,C 180,E1 -3689.999,E2 -3689.999} C_VEL
LIN {X 0,Y 544.545,Z 1015.187,A -85,B 0,C 180,E1 -3691.478,E2 -3691.478} C_VEL
LIN {X 0,Y 544.65,Z 1012.812,A -85,B 0,C 180,E1 -3692.957,E2 -3692.957} C_VEL
LIN {X 0,Y 544.683,Z 1009.899,A -85,B 0,C 180,E1 -3694.068,E2 -3694.068} C_VEL
LIN {X 0,Y 544.653,Z 1005.953,A -85,B 0,C 180,E1 -3695.181,E2 -3695.181} C_VEL
LIN {X 0,Y 544.73,Z 1000.639,A -85,B 0,C 180,E1 -3696.341,E2 -3696.341} C_VEL
LIN {X 0,Y 544.858,Z 993.244,A -85,B 0,C 180,E1 -3697.596,E2 -3697.596} C_VEL
LIN {X 0,Y 545.022,Z 985,A -85,B 0,C 180,E1 -3698.714,E2 -3698.714} C_VEL
LIN {X 0,Y 545.201,Z 976.551,A -85,B 0,C 180,E1 -3699.646,E2 -3699.646} C_VEL
LIN {X 0,Y 545.387,Z 966.111,A -85,B 0,C 180,E1 -3700.58,E2 -3700.58} C_VEL
LIN {X 0,Y 545.635,Z 954.373,A -85,B 0,C 180,E1 -3701.419,E2 -3701.419} C_VEL
LIN {X 0,Y 545.851,Z 942.514,A -85,B 0,C 180,E1 -3702.076,E2 -3702.076} C_VEL
LIN {X 0,Y 545.998,Z 930.202,A -85,B 0,C 180,E1 -3702.591,E2 -3702.591} C_VEL
LIN {X 0,Y 546.153,Z 917.565,A -85,B 0,C 180,E1 -3702.966,E2 -3702.966} C_VEL
LIN {X 0,Y 546.276,Z 904.402,A -85,B 0,C 180,E1 -3703.199,E2 -3703.199} C_VEL
LIN {X 0,Y 546.459,Z 808.19,A -85,B 0,C 180,E1 -3704.47,E2 -3704.47} C_VEL
LIN {X 0,Y 545.62,Z 802.04,A -85,B 0,C 180,E1 -3704.587,E2 -3704.587} C_VEL
LIN {X 0,Y 545.97,Z 780.32,A -85,B 0,C 180,E1 -3707.027,E2 -3707.027} C_VEL
LIN {X 0,Y 546.51,Z 754.329,A -85,B 0,C 180,E1 -3710.014,E2 -3710.014} C_VEL
LIN {X 0,Y 547.03,Z 729.89,A -85,B 0,C 180,E1 -3712.868,E2 -3712.868} C_VEL
LIN {X 0,Y 547.383,Z 712.459,A -85,B 0,C 180,E1 -3714.864,E2 -3714.864} C_VEL
LIN {X 0,Y 547.643,Z 696.441,A -85,B 0,C 180,E1 -3716.688,E2 -3716.688} C_VEL
LIN {X 0,Y 546.416,Z 690.323,A -85,B 0,C 180,E1 -3717.442,E2 -3717.442} C_VEL
LIN {X 0,Y 545.133,Z 684.698,A -85,B 0,C 180,E1 -3718.201,E2 -3718.201} C_VEL
LIN {X 0,Y 545.062,Z 684.587,A -85,B 0,C 180,E1 -3721.047,E2 -3721.047} C_VEL
LIN {X 0,Y 545.059,Z 684.587,A -85,B 0,C 180,E1 -3723.671,E2 -3723.671} C_VEL
LIN {X 0,Y 545.064,Z 684.588,A -85,B 0,C 180,E1 -3726.925,E2 -3726.925} C_VEL
LIN {X 0,Y 545.059,Z 684.589,A -85,B 0,C 180,E1 -3730.141,E2 -3730.141} C_VEL
LIN {X 0,Y 545.071,Z 684.586,A -85,B 0,C 180,E1 -3733.105,E2 -3733.105} C_VEL
LIN {X 0,Y 545.059,Z 684.585,A -85,B 0,C 180,E1 -3736.223,E2 -3736.223} C_VEL
LIN {X 0,Y 545.089,Z 684.589,A -85,B 0,C 180,E1 -3738.886,E2 -3738.886} C_VEL
LIN {X 0,Y 545.046,Z 684.586,A -85,B 0,C 180,E1 -3741.762,E2 -3741.762} C_VEL
LIN {X 0,Y 545.056,Z 684.584,A -85,B 0,C 180,E1 -3744.533,E2 -3744.533} C_VEL
LIN {X 0,Y 545.071,Z 684.593,A -85,B 0,C 180,E1 -3747.212,E2 -3747.212} C_VEL
LIN {X 0,Y 545.092,Z 684.583,A -85,B 0,C 180,E1 -3749.812,E2 -3749.812} C_VEL
LIN {X 0,Y 545.091,Z 684.582,A -85,B 0,C 180,E1 -3752.824,E2 -3752.824} C_VEL
LIN {X 0,Y 545.042,Z 684.594,A -85,B 0,C 180,E1 -3755.63,E2 -3755.63} C_VEL
LIN {X 0,Y 545.054,Z 684.584,A -85,B 0,C 180,E1 -3758.836,E2 -3758.836} C_VEL
LIN {X 0,Y 545.07,Z 684.585,A -85,B 0,C 180,E1 -3761.195,E2 -3761.195} C_VEL
LIN {X 0,Y 545.06,Z 684.588,A -85,B 0,C 180,E1 -3763.521,E2 -3763.521} C_VEL
LIN {X 0,Y 545.083,Z 684.59,A -85,B 0,C 180,E1 -3765.82,E2 -3765.82} C_VEL
LIN {X 0,Y 545.105,Z 684.578,A -85,B 0,C 180,E1 -3768.849,E2 -3768.849} C_VEL
LIN {X 0,Y 545.119,Z 684.581,A -85,B 0,C 180,E1 -3771.847,E2 -3771.847} C_VEL
LIN {X 0,Y 545.194,Z 684.567,A -85,B 0,C 180,E1 -3774.823,E2 -3774.823} C_VEL
LIN {X 0,Y 545.179,Z 684.571,A -85,B 0,C 180,E1 -3777.784,E2 -3777.784} C_VEL
LIN {X 0,Y 545.206,Z 684.57,A -85,B 0,C 180,E1 -3780.739,E2 -3780.739} C_VEL
LIN {X 0,Y 545.165,Z 684.573,A -85,B 0,C 180,E1 -3782.956,E2 -3782.956} C_VEL
LIN {X 0,Y 545.156,Z 684.573,A -85,B 0,C 180,E1 -3785.92,E2 -3785.92} C_VEL
LIN {X 0,Y 545.11,Z 684.584,A -85,B 0,C 180,E1 -3788.9,E2 -3788.9} C_VEL
LIN {X 0,Y 545.124,Z 684.575,A -85,B 0,C 180,E1 -3791.905,E2 -3791.905} C_VEL
LIN {X 0,Y 545.074,Z 684.591,A -85,B 0,C 180,E1 -3794.944,E2 -3794.944} C_VEL
LIN {X 0,Y 545.059,Z 684.584,A -85,B 0,C 180,E1 -3798.027,E2 -3798.027} C_VEL
LIN {X 0,Y 545.083,Z 684.582,A -85,B 0,C 180,E1 -3800.373,E2 -3800.373} C_VEL
LIN {X 0,Y 545.068,Z 684.585,A -85,B 0,C 180,E1 -3803.56,E2 -3803.56} C_VEL
LIN {X 0,Y 545.061,Z 684.585,A -85,B 0,C 180,E1 -3806.002,E2 -3806.002} C_VEL
LIN {X 0,Y 545.064,Z 684.582,A -85,B 0,C 180,E1 -3808.746,E2 -3808.746} C_VEL
LIN {X 0,Y 545.049,Z 684.591,A -85,B 0,C 180,E1 -3811.68,E2 -3811.68} C_VEL
LIN {X 0,Y 545.067,Z 684.584,A -85,B 0,C 180,E1 -3814.564,E2 -3814.564} C_VEL
LIN {X 0,Y 545.054,Z 684.586,A -85,B 0,C 180,E1 -3817.02,E2 -3817.02} C_VEL
LIN {X 0,Y 544.347,Z 684.683,A -85,B 0,C 180,E1 -3817.636,E2 -3817.636} C_VEL
LIN {X 0,Y 541.481,Z 685.04,A -85,B 0,C 180,E1 -3818.637,E2 -3818.637} C_VEL
LIN {X 0,Y 539.094,Z 685.336,A -85,B 0,C 180,E1 -3819.443,E2 -3819.443} C_VEL
LIN {X 0,Y 538.085,Z 685.46,A -85,B 0,C 180,E1 -3820.065,E2 -3820.065} C_VEL
LIN {X 0,Y 538.01,Z 685.465,A -85,B 0,C 180,E1 -3820.276,E2 -3820.276} C_VEL
LIN {X 0,Y 538.019,Z 685.462,A -85,B 0,C 180,E1 -3822.989,E2 -3822.989} C_VEL
LIN {X 0,Y 537.997,Z 685.469,A -85,B 0,C 180,E1 -3826.185,E2 -3826.185} C_VEL
LIN {X 0,Y 538.042,Z 685.462,A -85,B 0,C 180,E1 -3829.254,E2 -3829.254} C_VEL
LIN {X 0,Y 538.062,Z 685.626,A -85,B 0,C 180,E1 -3830.561,E2 -3830.561} C_VEL
LIN {X 0,Y 538.263,Z 686.582,A -85,B 0,C 180,E1 -3830.68,E2 -3830.68} C_VEL
LIN {X 0,Y 539.69,Z 690.75,A -85,B 0,C 180,E1 -3830.79,E2 -3830.79} C_VEL
LIN {X 0,Y 539.38,Z 765.265,A -85,B 0,C 180,E1 -3831.809,E2 -3831.809} C_VEL
LIN {X 0,Y 539.278,Z 778.725,A -85,B 0,C 180,E1 -3832.156,E2 -3832.156} C_VEL
LIN {X 0,Y 539.111,Z 790.077,A -85,B 0,C 180,E1 -3832.586,E2 -3832.586} C_VEL
LIN {X 0,Y 538.947,Z 801.147,A -85,B 0,C 180,E1 -3833.142,E2 -3833.142} C_VEL
LIN {X 0,Y 538.752,Z 812.828,A -85,B 0,C 180,E1 -3833.906,E2 -3833.906} C_VEL
LIN {X 0,Y 538.495,Z 822.852,A -85,B 0,C 180,E1 -3834.726,E2 -3834.726} C_VEL
LIN {X 0,Y 538.271,Z 832.287,A -85,B 0,C 180,E1 -3835.677,E2 -3835.677} C_VEL
LIN {X 0,Y 538.027,Z 840.715,A -85,B 0,C 180,E1 -3836.729,E2 -3836.729} C_VEL
LIN {X 0,Y 537.897,Z 848.352,A -85,B 0,C 180,E1 -3837.918,E2 -3837.918} C_VEL
LIN {X 0,Y 537.764,Z 853.563,A -85,B 0,C 180,E1 -3838.922,E2 -3838.922} C_VEL
LIN {X 0,Y 537.659,Z 858.875,A -85,B 0,C 180,E1 -3840.219,E2 -3840.219} C_VEL
LIN {X 0,Y 537.635,Z 861.758,A -85,B 0,C 180,E1 -3841.144,E2 -3841.144} C_VEL
LIN {X 0,Y 537.599,Z 863.708,A -85,B 0,C 180,E1 -3841.927,E2 -3841.927} C_VEL
LIN {X 0,Y 537.551,Z 865.286,A -85,B 0,C 180,E1 -3842.77,E2 -3842.77} C_VEL
LIN {X 0,Y 537.544,Z 866.345,A -85,B 0,C 180,E1 -3843.608,E2 -3843.608} C_VEL
LIN {X 0,Y 537.537,Z 866.947,A -85,B 0,C 180,E1 -3844.441,E2 -3844.441} C_VEL
LIN {X 0,Y 537.511,Z 867.031,A -85,B 0,C 180,E1 -3845.268,E2 -3845.268} C_VEL
LIN {X 0,Y 537.535,Z 866.576,A -85,B 0,C 180,E1 -3846.237,E2 -3846.237} C_VEL
LIN {X 0,Y 537.551,Z 865.864,A -85,B 0,C 180,E1 -3846.909,E2 -3846.909} C_VEL
LIN {X 0,Y 537.562,Z 863.687,A -85,B 0,C 180,E1 -3848.164,E2 -3848.164} C_VEL
LIN {X 0,Y 537.674,Z 860.596,A -85,B 0,C 180,E1 -3849.335,E2 -3849.335} C_VEL
LIN {X 0,Y 537.744,Z 856.107,A -85,B 0,C 180,E1 -3850.578,E2 -3850.578} C_VEL
LIN {X 0,Y 537.862,Z 849.708,A -85,B 0,C 180,E1 -3851.922,E2 -3851.922} C_VEL
LIN {X 0,Y 537.995,Z 842.431,A -85,B 0,C 180,E1 -3853.106,E2 -3853.106} C_VEL
LIN {X 0,Y 538.231,Z 833.342,A -85,B 0,C 180,E1 -3854.281,E2 -3854.281} C_VEL
LIN {X 0,Y 538.439,Z 823.789,A -85,B 0,C 180,E1 -3855.271,E2 -3855.271} C_VEL
LIN {X 0,Y 538.661,Z 813.458,A -85,B 0,C 180,E1 -3856.13,E2 -3856.13} C_VEL
LIN {X 0,Y 538.902,Z 801.75,A -85,B 0,C 180,E1 -3856.905,E2 -3856.905} C_VEL
LIN {X 0,Y 539.115,Z 789.713,A -85,B 0,C 180,E1 -3857.513,E2 -3857.513} C_VEL
LIN {X 0,Y 539.278,Z 776.286,A -85,B 0,C 180,E1 -3858.005,E2 -3858.005} C_VEL
LIN {X 0,Y 539.413,Z 763.965,A -85,B 0,C 180,E1 -3858.303,E2 -3858.303} C_VEL
LIN {X 0,Y 539.58,Z 690.407,A -85,B 0,C 180,E1 -3859.305,E2 -3859.305} C_VEL
LIN {X 0,Y 538.217,Z 686.373,A -85,B 0,C 180,E1 -3859.42,E2 -3859.42} C_VEL
LIN {X 0,Y 538.035,Z 685.542,A -85,B 0,C 180,E1 -3859.559,E2 -3859.559} C_VEL
LIN {X 0,Y 538.042,Z 685.463,A -85,B 0,C 180,E1 -3862.496,E2 -3862.496} C_VEL
LIN {X 0,Y 538.124,Z 685.45,A -85,B 0,C 180,E1 -3864.756,E2 -3864.756} C_VEL
LIN {X 0,Y 538.163,Z 685.449,A -85,B 0,C 180,E1 -3867.756,E2 -3867.756} C_VEL
LIN {X 0,Y 538.162,Z 685.451,A -85,B 0,C 180,E1 -3870.001,E2 -3870.001} C_VEL
LIN {X 0,Y 538.113,Z 685.452,A -85,B 0,C 180,E1 -3872.996,E2 -3872.996} C_VEL
LIN {X 0,Y 538.083,Z 685.458,A -85,B 0,C 180,E1 -3875.999,E2 -3875.999} C_VEL
LIN {X 0,Y 538.028,Z 685.463,A -85,B 0,C 180,E1 -3879.019,E2 -3879.019} C_VEL
LIN {X 0,Y 538.015,Z 685.463,A -85,B 0,C 180,E1 -3882.065,E2 -3882.065} C_VEL
LIN {X 0,Y 538.044,Z 685.46,A -85,B 0,C 180,E1 -3885.145,E2 -3885.145} C_VEL
LIN {X 0,Y 538.003,Z 685.465,A -85,B 0,C 180,E1 -3888.272,E2 -3888.272} C_VEL
LIN {X 0,Y 538.012,Z 685.465,A -85,B 0,C 180,E1 -3890.653,E2 -3890.653} C_VEL
LIN {X 0,Y 538.009,Z 685.47,A -85,B 0,C 180,E1 -3893.073,E2 -3893.073} C_VEL
LIN {X 0,Y 537.973,Z 685.464,A -85,B 0,C 180,E1 -3895.656,E2 -3895.656} C_VEL
LIN {X 0,Y 537.976,Z 685.464,A -85,B 0,C 180,E1 -3898.055,E2 -3898.055} C_VEL
LIN {X 0,Y 537.993,Z 685.466,A -85,B 0,C 180,E1 -3900.63,E2 -3900.63} C_VEL
LIN {X 0,Y 538.005,Z 685.467,A -85,B 0,C 180,E1 -3903.275,E2 -3903.275} C_VEL
LIN {X 0,Y 537.957,Z 685.466,A -85,B 0,C 180,E1 -3906.009,E2 -3906.009} C_VEL
LIN {X 0,Y 537.974,Z 685.468,A -85,B 0,C 180,E1 -3908.835,E2 -3908.835} C_VEL
LIN {X 0,Y 537.969,Z 685.472,A -85,B 0,C 180,E1 -3911.871,E2 -3911.871} C_VEL
LIN {X 0,Y 537.99,Z 685.465,A -85,B 0,C 180,E1 -3914.865,E2 -3914.865} C_VEL
LIN {X 0,Y 537.965,Z 685.471,A -85,B 0,C 180,E1 -3917.208,E2 -3917.208} C_VEL
LIN {X 0,Y 537.974,Z 685.469,A -85,B 0,C 180,E1 -3920.424,E2 -3920.424} C_VEL
LIN {X 0,Y 537.935,Z 685.472,A -85,B 0,C 180,E1 -3923.059,E2 -3923.059} C_VEL
LIN {X 0,Y 537.995,Z 685.473,A -85,B 0,C 180,E1 -3925.825,E2 -3925.825} C_VEL
LIN {X 0,Y 537.995,Z 685.47,A -85,B 0,C 180,E1 -3928.497,E2 -3928.497} C_VEL
LIN {X 0,Y 537.991,Z 685.469,A -85,B 0,C 180,E1 -3931.095,E2 -3931.095} C_VEL
LIN {X 0,Y 538.004,Z 685.68,A -85,B 0,C 180,E1 -3932.611,E2 -3932.611} C_VEL
LIN {X 0,Y 538.306,Z 686.866,A -85,B 0,C 180,E1 -3932.734,E2 -3932.734} C_VEL
LIN {X 0,Y 539.582,Z 690.902,A -85,B 0,C 180,E1 -3932.827,E2 -3932.827} C_VEL
LIN {X 0,Y 539.318,Z 761.466,A -85,B 0,C 180,E1 -3933.786,E2 -3933.786} C_VEL
LIN {X 0,Y 539.155,Z 773.42,A -85,B 0,C 180,E1 -3934.072,E2 -3934.072} C_VEL
LIN {X 0,Y 538.991,Z 784.359,A -85,B 0,C 180,E1 -3934.452,E2 -3934.452} C_VEL
LIN {X 0,Y 538.807,Z 794.527,A -85,B 0,C 180,E1 -3934.918,E2 -3934.918} C_VEL
LIN {X 0,Y 538.579,Z 804.907,A -85,B 0,C 180,E1 -3935.519,E2 -3935.519} C_VEL
LIN {X 0,Y 538.439,Z 813.587,A -85,B 0,C 180,E1 -3936.132,E2 -3936.132} C_VEL
LIN {X 0,Y 538.221,Z 821.955,A -85,B 0,C 180,E1 -3936.836,E2 -3936.836} C_VEL
LIN {X 0,Y 538.04,Z 830.843,A -85,B 0,C 180,E1 -3937.74,E2 -3937.74} C_VEL
LIN {X 0,Y 537.927,Z 837.499,A -85,B 0,C 180,E1 -3938.542,E2 -3938.542} C_VEL
LIN {X 0,Y 537.747,Z 844.405,A -85,B 0,C 180,E1 -3939.537,E2 -3939.537} C_VEL
LIN {X 0,Y 537.678,Z 850.351,A -85,B 0,C 180,E1 -3940.579,E2 -3940.579} C_VEL
LIN {X 0,Y 537.584,Z 855.551,A -85,B 0,C 180,E1 -3941.714,E2 -3941.714} C_VEL
LIN {X 0,Y 537.555,Z 858.949,A -85,B 0,C 180,E1 -3942.633,E2 -3942.633} C_VEL
LIN {X 0,Y 537.528,Z 860.902,A -85,B 0,C 180,E1 -3943.283,E2 -3943.283} C_VEL
LIN {X 0,Y 537.429,Z 864.259,A -85,B 0,C 180,E1 -3944.838,E2 -3944.838} C_VEL
LIN {X 0,Y 537.489,Z 865.239,A -85,B 0,C 180,E1 -3945.615,E2 -3945.615} C_VEL
LIN {X 0,Y 537.476,Z 865.983,A -85,B 0,C 180,E1 -3947.156,E2 -3947.156} C_VEL
LIN {X 0,Y 537.474,Z 865.679,A -85,B 0,C 180,E1 -3947.923,E2 -3947.923} C_VEL
LIN {X 0,Y 537.495,Z 863.95,A -85,B 0,C 180,E1 -3949.452,E2 -3949.452} C_VEL
LIN {X 0,Y 537.537,Z 860.401,A -85,B 0,C 180,E1 -3950.973,E2 -3950.973} C_VEL
LIN {X 0,Y 537.574,Z 856.601,A -85,B 0,C 180,E1 -3952.11,E2 -3952.11} C_VEL
LIN {X 0,Y 537.674,Z 851.671,A -85,B 0,C 180,E1 -3953.244,E2 -3953.244} C_VEL
LIN {X 0,Y 537.757,Z 846.624,A -85,B 0,C 180,E1 -3954.187,E2 -3954.187} C_VEL
LIN {X 0,Y 537.834,Z 840.577,A -85,B 0,C 180,E1 -3955.127,E2 -3955.127} C_VEL
LIN {X 0,Y 537.934,Z 833.322,A -85,B 0,C 180,E1 -3956.067,E2 -3956.067} C_VEL
LIN {X 0,Y 538.106,Z 826.503,A -85,B 0,C 180,E1 -3956.818,E2 -3956.818} C_VEL
LIN {X 0,Y 538.326,Z 817.29,A -85,B 0,C 180,E1 -3957.662,E2 -3957.662} C_VEL
LIN {X 0,Y 538.492,Z 808.742,A -85,B 0,C 180,E1 -3958.317,E2 -3958.317} C_VEL
LIN {X 0,Y 538.706,Z 798.261,A -85,B 0,C 180,E1 -3958.972,E2 -3958.972} C_VEL
LIN {X 0,Y 538.948,Z 787.916,A -85,B 0,C 180,E1 -3959.486,E2 -3959.486} C_VEL
LIN {X 0,Y 539.103,Z 777.664,A -85,B 0,C 180,E1 -3959.883,E2 -3959.883} C_VEL
LIN {X 0,Y 539.244,Z 766.946,A -85,B 0,C 180,E1 -3960.187,E2 -3960.187} C_VEL
LIN {X 0,Y 539.364,Z 755.893,A -85,B 0,C 180,E1 -3960.396,E2 -3960.396} C_VEL
LIN {X 0,Y 539.465,Z 690.03,A -85,B 0,C 180,E1 -3961.278,E2 -3961.278} C_VEL
LIN {X 0,Y 538.249,Z 686.423,A -85,B 0,C 180,E1 -3961.379,E2 -3961.379} C_VEL
LIN {X 0,Y 538.076,Z 685.532,A -85,B 0,C 180,E1 -3961.52,E2 -3961.52} C_VEL
LIN {X 0,Y 538.14,Z 685.452,A -85,B 0,C 180,E1 -3962.994,E2 -3962.994} C_VEL
LIN {X 0,Y 538.117,Z 685.459,A -85,B 0,C 180,E1 -3965.997,E2 -3965.997} C_VEL
LIN {X 0,Y 538.059,Z 685.458,A -85,B 0,C 180,E1 -3969.018,E2 -3969.018} C_VEL
LIN {X 0,Y 538.071,Z 685.462,A -85,B 0,C 180,E1 -3972.063,E2 -3972.063} C_VEL
LIN {X 0,Y 538.052,Z 685.458,A -85,B 0,C 180,E1 -3975.144,E2 -3975.144} C_VEL
LIN {X 0,Y 538.029,Z 685.468,A -85,B 0,C 180,E1 -3978.27,E2 -3978.27} C_VEL
LIN {X 0,Y 538.044,Z 685.467,A -85,B 0,C 180,E1 -3980.651,E2 -3980.651} C_VEL
LIN {X 0,Y 538.007,Z 685.464,A -85,B 0,C 180,E1 -3983.888,E2 -3983.888} C_VEL
LIN {X 0,Y 538.042,Z 685.463,A -85,B 0,C 180,E1 -3986.367,E2 -3986.367} C_VEL
LIN {X 0,Y 538.037,Z 685.468,A -85,B 0,C 180,E1 -3988.933,E2 -3988.933} C_VEL
LIN {X 0,Y 538.016,Z 685.462,A -85,B 0,C 180,E1 -3991.887,E2 -3991.887} C_VEL
LIN {X 0,Y 538.015,Z 685.466,A -85,B 0,C 180,E1 -3994.617,E2 -3994.617} C_VEL
LIN {X 0,Y 538.01,Z 685.471,A -85,B 0,C 180,E1 -3997.169,E2 -3997.169} C_VEL
LIN {X 0,Y 538.027,Z 685.462,A -85,B 0,C 180,E1 -3999.797,E2 -3999.797} C_VEL
LIN {X 0,Y 538.025,Z 685.464,A -85,B 0,C 180,E1 -4002.786,E2 -4002.786} C_VEL
LIN {X 0,Y 538.024,Z 685.463,A -85,B 0,C 180,E1 -4005.926,E2 -4005.926} C_VEL
LIN {X 0,Y 538.036,Z 685.46,A -85,B 0,C 180,E1 -4008.226,E2 -4008.226} C_VEL
LIN {X 0,Y 538.016,Z 685.466,A -85,B 0,C 180,E1 -4011.169,E2 -4011.169} C_VEL
LIN {X 0,Y 537.995,Z 685.468,A -85,B 0,C 180,E1 -4014.089,E2 -4014.089} C_VEL
LIN {X 0,Y 538.037,Z 685.461,A -85,B 0,C 180,E1 -4016.727,E2 -4016.727} C_VEL
LIN {X 0,Y 538.033,Z 685.468,A -85,B 0,C 180,E1 -4019.556,E2 -4019.556} C_VEL
LIN {X 0,Y 538.076,Z 685.677,A -85,B 0,C 180,E1 -4021.606,E2 -4021.606} C_VEL
LIN {X 0,Y 540.811,Z 697.815,A -85,B 0,C 180,E1 -4023.174,E2 -4023.174} C_VEL
LIN {X 0,Y 540.321,Z 722.606,A -85,B 0,C 180,E1 -4026.051,E2 -4026.051} C_VEL
LIN {X 0,Y 539.821,Z 748.361,A -85,B 0,C 180,E1 -4029.02,E2 -4029.02} C_VEL
LIN {X 0,Y 539.146,Z 775.869,A -85,B 0,C 180,E1 -4032.232,E2 -4032.232} C_VEL
LIN {X 0,Y 538.678,Z 801.953,A -85,B 0,C 180,E1 -4035.216,E2 -4035.216} C_VEL
LIN {X 0,Y 539.703,Z 810.352,A -85,B 0,C 180,E1 -4035.374,E2 -4035.374} C_VEL
LIN {X 0,Y 539.315,Z 911.896,A -85,B 0,C 180,E1 -4036.745,E2 -4036.745} C_VEL
LIN {X 0,Y 539.181,Z 925.184,A -85,B 0,C 180,E1 -4037.077,E2 -4037.077} C_VEL
LIN {X 0,Y 538.953,Z 937.345,A -85,B 0,C 180,E1 -4037.526,E2 -4037.526} C_VEL
LIN {X 0,Y 538.79,Z 948.768,A -85,B 0,C 180,E1 -4038.095,E2 -4038.095} C_VEL
LIN {X 0,Y 538.556,Z 959.891,A -85,B 0,C 180,E1 -4038.806,E2 -4038.806} C_VEL
LIN {X 0,Y 538.295,Z 970.527,A -85,B 0,C 180,E1 -4039.657,E2 -4039.657} C_VEL
LIN {X 0,Y 538.068,Z 980.082,A -85,B 0,C 180,E1 -4040.602,E2 -4040.602} C_VEL
LIN {X 0,Y 537.915,Z 987.952,A -85,B 0,C 180,E1 -4041.547,E2 -4041.547} C_VEL
LIN {X 0,Y 537.756,Z 995.615,A -85,B 0,C 180,E1 -4042.678,E2 -4042.678} C_VEL
LIN {X 0,Y 537.696,Z 1002.674,A -85,B 0,C 180,E1 -4043.997,E2 -4043.997} C_VEL
LIN {X 0,Y 537.54,Z 1007.368,A -85,B 0,C 180,E1 -4045.124,E2 -4045.124} C_VEL
LIN {X 0,Y 537.591,Z 1010.955,A -85,B 0,C 180,E1 -4046.251,E2 -4046.251} C_VEL
LIN {X 0,Y 537.551,Z 1012.805,A -85,B 0,C 180,E1 -4047.001,E2 -4047.001} C_VEL
LIN {X 0,Y 537.489,Z 1014.194,A -85,B 0,C 180,E1 -4047.751,E2 -4047.751} C_VEL
LIN {X 0,Y 537.442,Z 1015.785,A -85,B 0,C 180,E1 -4049.25,E2 -4049.25} C_VEL
LIN {X 0,Y 537.442,Z 1016,A -85,B 0,C 180,E1 -4049.999,E2 -4049.999} C_VEL
LIN {X 0,Y 537.451,Z 1015.186,A -85,B 0,C 180,E1 -4051.498,E2 -4051.498} C_VEL
LIN {X 0,Y 537.489,Z 1014.199,A -85,B 0,C 180,E1 -4052.247,E2 -4052.247} C_VEL
LIN {X 0,Y 537.551,Z 1012.812,A -85,B 0,C 180,E1 -4052.997,E2 -4052.997} C_VEL
LIN {X 0,Y 537.603,Z 1009.899,A -85,B 0,C 180,E1 -4054.122,E2 -4054.122} C_VEL
LIN {X 0,Y 537.587,Z 1005.953,A -85,B 0,C 180,E1 -4055.249,E2 -4055.249} C_VEL
LIN {X 0,Y 537.645,Z 1001.12,A -85,B 0,C 180,E1 -4056.327,E2 -4056.327} C_VEL
LIN {X 0,Y 537.789,Z 994.475,A -85,B 0,C 180,E1 -4057.508,E2 -4057.508} C_VEL
LIN {X 0,Y 537.965,Z 986.487,A -85,B 0,C 180,E1 -4058.639,E2 -4058.639} C_VEL
LIN {X 0,Y 538.143,Z 978.346,A -85,B 0,C 180,E1 -4059.584,E2 -4059.584} C_VEL
LIN {X 0,Y 538.346,Z 968.413,A -85,B 0,C 180,E1 -4060.53,E2 -4060.53} C_VEL
LIN {X 0,Y 538.576,Z 958.607,A -85,B 0,C 180,E1 -4061.287,E2 -4061.287} C_VEL
LIN {X 0,Y 538.803,Z 947.718,A -85,B 0,C 180,E1 -4061.963,E2 -4061.963} C_VEL
LIN {X 0,Y 538.988,Z 935.134,A -85,B 0,C 180,E1 -4062.566,E2 -4062.566} C_VEL
LIN {X 0,Y 539.206,Z 922.134,A -85,B 0,C 180,E1 -4063.016,E2 -4063.016} C_VEL
LIN {X 0,Y 539.344,Z 909.183,A -85,B 0,C 180,E1 -4063.3,E2 -4063.3} C_VEL
LIN {X 0,Y 539.632,Z 809.118,A -85,B 0,C 180,E1 -4064.645,E2 -4064.645} C_VEL
LIN {X 0,Y 538.68,Z 802.061,A -85,B 0,C 180,E1 -4064.778,E2 -4064.778} C_VEL
LIN {X 0,Y 539.134,Z 777.264,A -85,B 0,C 180,E1 -4067.606,E2 -4067.606} C_VEL
LIN {X 0,Y 539.762,Z 750.062,A -85,B 0,C 180,E1 -4070.78,E2 -4070.78} C_VEL
LIN {X 0,Y 540.097,Z 731.023,A -85,B 0,C 180,E1 -4072.976,E2 -4072.976} C_VEL
LIN {X 0,Y 540.487,Z 709.757,A -85,B 0,C 180,E1 -4075.409,E2 -4075.409} C_VEL
LIN {X 0,Y 540.706,Z 697.291,A -85,B 0,C 180,E1 -4076.849,E2 -4076.849} C_VEL
LIN {X 0,Y 538.094,Z 685.636,A -85,B 0,C 180,E1 -4078.364,E2 -4078.364} C_VEL
LIN {X 0,Y 538.004,Z 685.467,A -85,B 0,C 180,E1 -4081.5,E2 -4081.5} C_VEL
LIN {X 0,Y 538.013,Z 685.467,A -85,B 0,C 180,E1 -4084.172,E2 -4084.172} C_VEL
LIN {X 0,Y 537.998,Z 685.466,A -85,B 0,C 180,E1 -4087.169,E2 -4087.169} C_VEL
LIN {X 0,Y 538.016,Z 685.463,A -85,B 0,C 180,E1 -4089.796,E2 -4089.796} C_VEL
LIN {X 0,Y 538.011,Z 685.469,A -85,B 0,C 180,E1 -4092.785,E2 -4092.785} C_VEL
LIN {X 0,Y 538.025,Z 685.464,A -85,B 0,C 180,E1 -4095.14,E2 -4095.14} C_VEL
LIN {X 0,Y 538.033,Z 685.461,A -85,B 0,C 180,E1 -4098.227,E2 -4098.227} C_VEL
LIN {X 0,Y 538.007,Z 685.47,A -85,B 0,C 180,E1 -4101.169,E2 -4101.169} C_VEL
LIN {X 0,Y 538.02,Z 685.458,A -85,B 0,C 180,E1 -4104.082,E2 -4104.082} C_VEL
LIN {X 0,Y 538.021,Z 685.464,A -85,B 0,C 180,E1 -4106.727,E2 -4106.727} C_VEL
LIN {X 0,Y 538.028,Z 685.466,A -85,B 0,C 180,E1 -4109.553,E2 -4109.553} C_VEL
LIN {X 0,Y 538.038,Z 685.46,A -85,B 0,C 180,E1 -4111.95,E2 -4111.95} C_VEL
LIN {X 0,Y 538.065,Z 685.455,A -85,B 0,C 180,E1 -4114.467,E2 -4114.467} C_VEL
LIN {X 0,Y 538.012,Z 685.464,A -85,B 0,C 180,E1 -4116.928,E2 -4116.928} C_VEL
LIN {X 0,Y 538.067,Z 685.458,A -85,B 0,C 180,E1 -4120.147,E2 -4120.147} C_VEL
LIN {X 0,Y 538.012,Z 685.463,A -85,B 0,C 180,E1 -4123.299,E2 -4123.299} C_VEL
LIN {X 0,Y 538.052,Z 685.464,A -85,B 0,C 180,E1 -4125.63,E2 -4125.63} C_VEL
LIN {X 0,Y 538.065,Z 685.456,A -85,B 0,C 180,E1 -4128.701,E2 -4128.701} C_VEL
LIN {X 0,Y 538.076,Z 685.456,A -85,B 0,C 180,E1 -4131.74,E2 -4131.74} C_VEL
LIN {X 0,Y 538.152,Z 685.445,A -85,B 0,C 180,E1 -4134.755,E2 -4134.755} C_VEL
LIN {X 0,Y 538.152,Z 685.447,A -85,B 0,C 180,E1 -4137.755,E2 -4137.755} C_VEL
LIN {X 0,Y 538.175,Z 685.445,A -85,B 0,C 180,E1 -4140.748,E2 -4140.748} C_VEL
LIN {X 0,Y 538.131,Z 685.449,A -85,B 0,C 180,E1 -4142.995,E2 -4142.995} C_VEL
LIN {X 0,Y 538.107,Z 685.451,A -85,B 0,C 180,E1 -4145.998,E2 -4145.998} C_VEL
LIN {X 0,Y 538.061,Z 685.46,A -85,B 0,C 180,E1 -4149.018,E2 -4149.018} C_VEL
LIN {X 0,Y 538.072,Z 685.455,A -85,B 0,C 180,E1 -4152.063,E2 -4152.063} C_VEL
LIN {X 0,Y 538.033,Z 685.464,A -85,B 0,C 180,E1 -4155.144,E2 -4155.144} C_VEL
LIN {X 0,Y 538.014,Z 685.463,A -85,B 0,C 180,E1 -4158.271,E2 -4158.271} C_VEL
LIN {X 0,Y 538.028,Z 685.463,A -85,B 0,C 180,E1 -4160.652,E2 -4160.652} C_VEL
LIN {X 0,Y 537.987,Z 685.464,A -85,B 0,C 180,E1 -4163.889,E2 -4163.889} C_VEL
LIN {X 0,Y 538.027,Z 685.461,A -85,B 0,C 180,E1 -4166.368,E2 -4166.368} C_VEL
